LIN {X 0,Y 418.31,Z 399.821,A -85,B 0,C 180,E1 -10290.267,E2 -10290.267} C_VEL
LIN {X 0,Y 417.846,Z 405.193,A -85,B 0,C 180,E1 -10291.993,E2 -10291.993} C_VEL
LIN {X 0,Y 417.536,Z 409.039,A -85,B 0,C 180,E1 -10293.742,E2 -10293.742} C_VEL
LIN {X 0,Y 417.376,Z 410.854,A -85,B 0,C 180,E1 -10294.925,E2 -10294.925} C_VEL
LIN {X 0,Y 417.277,Z 412.013,A -85,B 0,C 180,E1 -10296.121,E2 -10296.121} C_VEL
LIN {X 0,Y 417.19,Z 412.615,A -85,B 0,C 180,E1 -10297.65,E2 -10297.65} C_VEL
LIN {X 0,Y 417.218,Z 412.19,A -85,B 0,C 180,E1 -10299.207,E2 -10299.207} C_VEL
LIN {X 0,Y 417.254,Z 410.33,A -85,B 0,C 180,E1 -10301.064,E2 -10301.064} C_VEL
LIN {X 0,Y 417.561,Z 406.754,A -85,B 0,C 180,E1 -10302.973,E2 -10302.973} C_VEL
LIN {X 0,Y 417.802,Z 402.306,A -85,B 0,C 180,E1 -10304.611,E2 -10304.611} C_VEL
LIN {X 0,Y 418.147,Z 396.207,A -85,B 0,C 180,E1 -10306.28,E2 -10306.28} C_VEL
LIN {X 0,Y 418.601,Z 389.043,A -85,B 0,C 180,E1 -10307.812,E2 -10307.812} C_VEL
LIN {X 0,Y 419.168,Z 381.176,A -85,B 0,C 180,E1 -10309.164,E2 -10309.164} C_VEL
LIN {X 0,Y 419.798,Z 371.573,A -85,B 0,C 180,E1 -10310.493,E2 -10310.493} C_VEL
LIN {X 0,Y 420.433,Z 361.16,A -85,B 0,C 180,E1 -10311.657,E2 -10311.657} C_VEL
LIN {X 0,Y 421.113,Z 349.41,A -85,B 0,C 180,E1 -10312.698,E2 -10312.698} C_VEL
LIN {X 0,Y 421.702,Z 337.687,A -85,B 0,C 180,E1 -10313.505,E2 -10313.505} C_VEL
LIN {X 0,Y 422.117,Z 325.639,A -85,B 0,C 180,E1 -10314.137,E2 -10314.137} C_VEL
LIN {X 0,Y 422.396,Z 313.572,A -85,B 0,C 180,E1 -10314.588,E2 -10314.588} C_VEL
LIN {X 0,Y 422.59,Z 300.07,A -85,B 0,C 180,E1 -10314.896,E2 -10314.896} C_VEL
LIN {X 0,Y 423.699,Z 218.43,A -85,B 0,C 180,E1 -10316.385,E2 -10316.385} C_VEL
LIN {X 0,Y 418.788,Z 204.246,A -85,B 0,C 180,E1 -10316.864,E2 -10316.864} C_VEL
LIN {X 0,Y 418.263,Z 202.387,A -85,B 0,C 180,E1 -10316.944,E2 -10316.944} C_VEL
LIN {X 0,Y 418.244,Z 202.385,A -85,B 0,C 180,E1 -10319.728,E2 -10319.728} C_VEL
LIN {X 0,Y 418.305,Z 202.381,A -85,B 0,C 180,E1 -10323.023,E2 -10323.023} C_VEL
LIN {X 0,Y 418.273,Z 202.379,A -85,B 0,C 180,E1 -10326.218,E2 -10326.218} C_VEL
LIN {X 0,Y 418.232,Z 202.385,A -85,B 0,C 180,E1 -10328.246,E2 -10328.246} C_VEL
LIN {X 0,Y 417.595,Z 202.47,A -85,B 0,C 180,E1 -10329.05,E2 -10329.05} C_VEL
LIN {X 0,Y 414.761,Z 202.818,A -85,B 0,C 180,E1 -10330.357,E2 -10330.357} C_VEL
LIN {X 0,Y 412.349,Z 203.119,A -85,B 0,C 180,E1 -10331.413,E2 -10331.413} C_VEL
LIN {X 0,Y 411.316,Z 203.246,A -85,B 0,C 180,E1 -10332.229,E2 -10332.229} C_VEL
LIN {X 0,Y 411.235,Z 203.256,A -85,B 0,C 180,E1 -10332.505,E2 -10332.505} C_VEL
LIN {X 0,Y 411.26,Z 203.256,A -85,B 0,C 180,E1 -10335.148,E2 -10335.148} C_VEL
LIN {X 0,Y 411.285,Z 203.251,A -85,B 0,C 180,E1 -10338.168,E2 -10338.168} C_VEL
LIN {X 0,Y 411.32,Z 203.248,A -85,B 0,C 180,E1 -10341.154,E2 -10341.154} C_VEL
LIN {X 0,Y 411.445,Z 203.231,A -85,B 0,C 180,E1 -10344.118,E2 -10344.118} C_VEL
LIN {X 0,Y 411.511,Z 203.223,A -85,B 0,C 180,E1 -10348.043,E2 -10348.043} C_VEL
LIN {X 0,Y 411.637,Z 203.208,A -85,B 0,C 180,E1 -10350,E2 -10350} C_VEL
LIN {X 0,Y 411.446,Z 203.231,A -85,B 0,C 180,E1 -10352.938,E2 -10352.938} C_VEL
LIN {X 0,Y 411.425,Z 203.234,A -85,B 0,C 180,E1 -10356.868,E2 -10356.868} C_VEL
LIN {X 0,Y 411.293,Z 203.251,A -85,B 0,C 180,E1 -10359.839,E2 -10359.839} C_VEL
LIN {X 0,Y 411.307,Z 203.247,A -85,B 0,C 180,E1 -10363.104,E2 -10363.104} C_VEL
LIN {X 0,Y 411.259,Z 203.253,A -85,B 0,C 180,E1 -10366.889,E2 -10366.889} C_VEL
LIN {X 0,Y 411.233,Z 203.263,A -85,B 0,C 180,E1 -10369.987,E2 -10369.987} C_VEL
LIN {X 0,Y 411.197,Z 203.261,A -85,B 0,C 180,E1 -10373.148,E2 -10373.148} C_VEL
LIN {X 0,Y 411.197,Z 203.262,A -85,B 0,C 180,E1 -10376.384,E2 -10376.384} C_VEL
LIN {X 0,Y 411.2,Z 203.266,A -85,B 0,C 180,E1 -10379.713,E2 -10379.713} C_VEL
LIN {X 0,Y 411.209,Z 203.261,A -85,B 0,C 180,E1 -10383.156,E2 -10383.156} C_VEL
LIN {X 0,Y 411.194,Z 203.261,A -85,B 0,C 180,E1 -10386.553,E2 -10386.553} C_VEL
LIN {X 0,Y 411.194,Z 203.266,A -85,B 0,C 180,E1 -10389.724,E2 -10389.724} C_VEL
LIN {X 0,Y 411.172,Z 203.267,A -85,B 0,C 180,E1 -10393.134,E2 -10393.134} C_VEL
LIN {X 0,Y 411.169,Z 203.266,A -85,B 0,C 180,E1 -10395.881,E2 -10395.881} C_VEL
LIN {X 0,Y 411.154,Z 203.267,A -85,B 0,C 180,E1 -10398.774,E2 -10398.774} C_VEL
LIN {X 0,Y 411.188,Z 203.262,A -85,B 0,C 180,E1 -10402.026,E2 -10402.026} C_VEL
LIN {X 0,Y 411.207,Z 203.261,A -85,B 0,C 180,E1 -10405.667,E2 -10405.667} C_VEL
LIN {X 0,Y 411.191,Z 203.268,A -85,B 0,C 180,E1 -10409.153,E2 -10409.153} C_VEL
LIN {X 0,Y 411.182,Z 203.265,A -85,B 0,C 180,E1 -10411.407,E2 -10411.407} C_VEL
LIN {X 0,Y 411.229,Z 203.264,A -85,B 0,C 180,E1 -10414.93,E2 -10414.93} C_VEL
LIN {X 0,Y 411.207,Z 203.259,A -85,B 0,C 180,E1 -10417.914,E2 -10417.914} C_VEL
LIN {X 0,Y 411.222,Z 203.262,A -85,B 0,C 180,E1 -10421.051,E2 -10421.051} C_VEL
LIN {X 0,Y 411.256,Z 203.254,A -85,B 0,C 180,E1 -10424.132,E2 -10424.132} C_VEL
LIN {X 0,Y 411.306,Z 203.249,A -85,B 0,C 180,E1 -10427.166,E2 -10427.166} C_VEL
LIN {X 0,Y 411.293,Z 203.251,A -85,B 0,C 180,E1 -10430.161,E2 -10430.161} C_VEL
LIN {X 0,Y 411.396,Z 203.237,A -85,B 0,C 180,E1 -10433.132,E2 -10433.132} C_VEL
LIN {X 0,Y 411.301,Z 203.249,A -85,B 0,C 180,E1 -10435.099,E2 -10435.099} C_VEL
LIN {X 0,Y 411.512,Z 203.224,A -85,B 0,C 180,E1 -10438.043,E2 -10438.043} C_VEL
LIN {X 0,Y 411.433,Z 203.232,A -85,B 0,C 180,E1 -10440.979,E2 -10440.979} C_VEL
LIN {X 0,Y 411.433,Z 203.232,A -85,B 0,C 180,E1 -10442.938,E2 -10442.938} C_VEL
LIN {X 0,Y 411.432,Z 203.234,A -85,B 0,C 180,E1 -10445.883,E2 -10445.883} C_VEL
LIN {X 0,Y 411.32,Z 203.246,A -85,B 0,C 180,E1 -10448.846,E2 -10448.846} C_VEL
LIN {X 0,Y 411.286,Z 203.254,A -85,B 0,C 180,E1 -10451.833,E2 -10451.833} C_VEL
LIN {X 0,Y 411.235,Z 203.256,A -85,B 0,C 180,E1 -10454.854,E2 -10454.854} C_VEL
LIN {X 0,Y 411.233,Z 203.263,A -85,B 0,C 180,E1 -10457.916,E2 -10457.916} C_VEL
LIN {X 0,Y 411.199,Z 203.26,A -85,B 0,C 180,E1 -10461.034,E2 -10461.034} C_VEL
LIN {X 0,Y 411.195,Z 203.263,A -85,B 0,C 180,E1 -10464.218,E2 -10464.218} C_VEL
LIN {X 0,Y 411.175,Z 203.268,A -85,B 0,C 180,E1 -10467.484,E2 -10467.484} C_VEL
LIN {X 0,Y 411.2,Z 203.267,A -85,B 0,C 180,E1 -10469.713,E2 -10469.713} C_VEL
LIN {X 0,Y 411.207,Z 203.262,A -85,B 0,C 180,E1 -10473.156,E2 -10473.156} C_VEL
LIN {X 0,Y 411.194,Z 203.261,A -85,B 0,C 180,E1 -10476.552,E2 -10476.552} C_VEL
LIN {X 0,Y 411.172,Z 203.267,A -85,B 0,C 180,E1 -10479.72,E2 -10479.72} C_VEL
LIN {X 0,Y 411.165,Z 203.269,A -85,B 0,C 180,E1 -10483.135,E2 -10483.135} C_VEL
LIN {X 0,Y 411.166,Z 203.266,A -85,B 0,C 180,E1 -10485.882,E2 -10485.882} C_VEL
LIN {X 0,Y 411.165,Z 203.268,A -85,B 0,C 180,E1 -10489.493,E2 -10489.493} C_VEL
LIN {X 0,Y 411.19,Z 203.262,A -85,B 0,C 180,E1 -10492.025,E2 -10492.025} C_VEL
LIN {X 0,Y 411.195,Z 203.263,A -85,B 0,C 180,E1 -10495.665,E2 -10495.665} C_VEL
LIN {X 0,Y 411.191,Z 203.267,A -85,B 0,C 180,E1 -10499.152,E2 -10499.152} C_VEL
LIN {X 0,Y 411.262,Z 203.344,A -85,B 0,C 180,E1 -10500.374,E2 -10500.374} C_VEL
LIN {X 0,Y 414.279,Z 218.043,A -85,B 0,C 180,E1 -10503.284,E2 -10503.284} C_VEL
LIN {X 0,Y 414.784,Z 222.006,A -85,B 0,C 180,E1 -10504.037,E2 -10504.037} C_VEL
LIN {X 0,Y 413.508,Z 241.529,A -85,B 0,C 180,E1 -10507.517,E2 -10507.517} C_VEL
LIN {X 0,Y 412.396,Z 260.082,A -85,B 0,C 180,E1 -10510.784,E2 -10510.784} C_VEL
LIN {X 0,Y 416.32,Z 291.809,A -85,B 0,C 180,E1 -10511.587,E2 -10511.587} C_VEL
LIN {X 0,Y 415.21,Z 369.766,A -85,B 0,C 180,E1 -10513.055,E2 -10513.055} C_VEL
LIN {X 0,Y 414.703,Z 383.404,A -85,B 0,C 180,E1 -10513.509,E2 -10513.509} C_VEL
LIN {X 0,Y 414.037,Z 395.804,A -85,B 0,C 180,E1 -10514.114,E2 -10514.114} C_VEL
LIN {X 0,Y 413.33,Z 406.944,A -85,B 0,C 180,E1 -10514.845,E2 -10514.845} C_VEL
LIN {X 0,Y 412.607,Z 417.276,A -85,B 0,C 180,E1 -10515.701,E2 -10515.701} C_VEL
LIN {X 0,Y 411.914,Z 428.377,A -85,B 0,C 180,E1 -10516.85,E2 -10516.85} C_VEL
LIN {X 0,Y 411.315,Z 438.558,A -85,B 0,C 180,E1 -10518.168,E2 -10518.168} C_VEL
LIN {X 0,Y 410.671,Z 447.696,A -85,B 0,C 180,E1 -10519.648,E2 -10519.648} C_VEL
LIN {X 0,Y 410.341,Z 455.065,A -85,B 0,C 180,E1 -10521.133,E2 -10521.133} C_VEL
LIN {X 0,Y 410.171,Z 460.941,A -85,B 0,C 180,E1 -10522.616,E2 -10522.616} C_VEL
LIN {X 0,Y 410.066,Z 465.54,A -85,B 0,C 180,E1 -10524.097,E2 -10524.097} C_VEL
LIN {X 0,Y 410.102,Z 467.957,A -85,B 0,C 180,E1 -10525.084,E2 -10525.084} C_VEL
LIN {X 0,Y 410.061,Z 469.921,A -85,B 0,C 180,E1 -10526.069,E2 -10526.069} C_VEL
LIN {X 0,Y 410.17,Z 471.461,A -85,B 0,C 180,E1 -10527.053,E2 -10527.053} C_VEL
LIN {X 0,Y 410.173,Z 472.52,A -85,B 0,C 180,E1 -10528.036,E2 -10528.036} C_VEL
LIN {X 0,Y 410.163,Z 473.165,A -85,B 0,C 180,E1 -10529.018,E2 -10529.018} C_VEL
LIN {X 0,Y 410.14,Z 473.407,A -85,B 0,C 180,E1 -10530,E2 -10530} C_VEL
LIN {X 0,Y 410.163,Z 473.239,A -85,B 0,C 180,E1 -10530.982,E2 -10530.982} C_VEL
LIN {X 0,Y 410.15,Z 472.618,A -85,B 0,C 180,E1 -10531.964,E2 -10531.964} C_VEL
LIN {X 0,Y 410.174,Z 471.595,A -85,B 0,C 180,E1 -10532.946,E2 -10532.946} C_VEL
LIN {X 0,Y 410.06,Z 470.15,A -85,B 0,C 180,E1 -10533.931,E2 -10533.931} C_VEL
LIN {X 0,Y 410.08,Z 467.14,A -85,B 0,C 180,E1 -10535.408,E2 -10535.408} C_VEL
LIN {X 0,Y 410.162,Z 463.07,A -85,B 0,C 180,E1 -10536.889,E2 -10536.889} C_VEL
LIN {X 0,Y 410.336,Z 456.838,A -85,B 0,C 180,E1 -10538.619,E2 -10538.619} C_VEL
LIN {X 0,Y 410.617,Z 450.013,A -85,B 0,C 180,E1 -10540.104,E2 -10540.104} C_VEL
LIN {X 0,Y 411.22,Z 441.574,A -85,B 0,C 180,E1 -10541.584,E2 -10541.584} C_VEL
LIN {X 0,Y 411.787,Z 432.967,A -85,B 0,C 180,E1 -10542.819,E2 -10542.819} C_VEL
LIN {X 0,Y 412.572,Z 422.411,A -85,B 0,C 180,E1 -10544.048,E2 -10544.048} C_VEL
LIN {X 0,Y 413.448,Z 410.573,A -85,B 0,C 180,E1 -10545.15,E2 -10545.15} C_VEL
LIN {X 0,Y 414.331,Z 398.849,A -85,B 0,C 180,E1 -10546,E2 -10546} C_VEL
LIN {X 0,Y 415.062,Z 386.782,A -85,B 0,C 180,E1 -10546.666,E2 -10546.666} C_VEL
LIN {X 0,Y 415.84,Z 372.978,A -85,B 0,C 180,E1 -10547.203,E2 -10547.203} C_VEL
LIN {X 0,Y 416.177,Z 358.822,A -85,B 0,C 180,E1 -10547.537,E2 -10547.537} C_VEL
LIN {X 0,Y 417.102,Z 289.747,A -85,B 0,C 180,E1 -10548.852,E2 -10548.852} C_VEL
LIN {X 0,Y 414.27,Z 267.739,A -85,B 0,C 180,E1 -10549.447,E2 -10549.447} C_VEL
LIN {X 0,Y 412.657,Z 257.23,A -85,B 0,C 180,E1 -10549.78,E2 -10549.78} C_VEL
LIN {X 0,Y 413.871,Z 235.468,A -85,B 0,C 180,E1 -10553.511,E2 -10553.511} C_VEL
LIN {X 0,Y 414.745,Z 220.411,A -85,B 0,C 180,E1 -10556.141,E2 -10556.141} C_VEL
LIN {X 0,Y 412.639,Z 209.36,A -85,B 0,C 180,E1 -10558.274,E2 -10558.274} C_VEL
LIN {X 0,Y 411.211,Z 203.268,A -85,B 0,C 180,E1 -10559.54,E2 -10559.54} C_VEL
LIN {X 0,Y 411.207,Z 203.265,A -85,B 0,C 180,E1 -10563.155,E2 -10563.155} C_VEL
LIN {X 0,Y 411.192,Z 203.267,A -85,B 0,C 180,E1 -10566.552,E2 -10566.552} C_VEL
LIN {X 0,Y 411.17,Z 203.266,A -85,B 0,C 180,E1 -10569.72,E2 -10569.72} C_VEL
LIN {X 0,Y 411.17,Z 203.266,A -85,B 0,C 180,E1 -10573.134,E2 -10573.134} C_VEL
LIN {X 0,Y 411.167,Z 203.265,A -85,B 0,C 180,E1 -10575.881,E2 -10575.881} C_VEL
LIN {X 0,Y 411.155,Z 203.27,A -85,B 0,C 180,E1 -10578.773,E2 -10578.773} C_VEL
LIN {X 0,Y 411.186,Z 203.266,A -85,B 0,C 180,E1 -10582.025,E2 -10582.025} C_VEL
LIN {X 0,Y 411.205,Z 203.26,A -85,B 0,C 180,E1 -10585.666,E2 -10585.666} C_VEL
LIN {X 0,Y 411.189,Z 203.263,A -85,B 0,C 180,E1 -10589.152,E2 -10589.152} C_VEL
LIN {X 0,Y 411.189,Z 203.263,A -85,B 0,C 180,E1 -10592.517,E2 -10592.517} C_VEL
LIN {X 0,Y 411.211,Z 203.264,A -85,B 0,C 180,E1 -10595.784,E2 -10595.784} C_VEL
LIN {X 0,Y 411.196,Z 203.261,A -85,B 0,C 180,E1 -10598.966,E2 -10598.966} C_VEL
LIN {X 0,Y 411.245,Z 203.256,A -85,B 0,C 180,E1 -10602.084,E2 -10602.084} C_VEL
LIN {X 0,Y 411.258,Z 203.254,A -85,B 0,C 180,E1 -10605.147,E2 -10605.147} C_VEL
LIN {X 0,Y 411.283,Z 203.25,A -85,B 0,C 180,E1 -10608.167,E2 -10608.167} C_VEL
LIN {X 0,Y 411.44,Z 203.233,A -85,B 0,C 180,E1 -10612.189,E2 -10612.189} C_VEL
LIN {X 0,Y 411.471,Z 203.229,A -85,B 0,C 180,E1 -10614.118,E2 -10614.118} C_VEL
LIN {X 0,Y 411.51,Z 203.223,A -85,B 0,C 180,E1 -10618.042,E2 -10618.042} C_VEL
LIN {X 0,Y 411.64,Z 203.208,A -85,B 0,C 180,E1 -10620,E2 -10620} C_VEL
LIN {X 0,Y 411.458,Z 203.233,A -85,B 0,C 180,E1 -10622.937,E2 -10622.937} C_VEL
LIN {X 0,Y 411.424,Z 203.237,A -85,B 0,C 180,E1 -10626.868,E2 -10626.868} C_VEL
LIN {X 0,Y 411.291,Z 203.254,A -85,B 0,C 180,E1 -10629.839,E2 -10629.839} C_VEL
LIN {X 0,Y 411.305,Z 203.258,A -85,B 0,C 180,E1 -10633.104,E2 -10633.104} C_VEL
LIN {X 0,Y 411.302,Z 203.255,A -85,B 0,C 180,E1 -10636.887,E2 -10636.887} C_VEL
LIN {X 0,Y 411.275,Z 203.368,A -85,B 0,C 180,E1 -10638.089,E2 -10638.089} C_VEL
LIN {X 0,Y 411.383,Z 204.007,A -85,B 0,C 180,E1 -10638.23,E2 -10638.23} C_VEL
LIN {X 0,Y 418.004,Z 220.696,A -85,B 0,C 180,E1 -10638.962,E2 -10638.962} C_VEL
LIN {X 0,Y 418.199,Z 223.122,A -85,B 0,C 180,E1 -10639.023,E2 -10639.023} C_VEL
LIN {X 0,Y 416.618,Z 312.115,A -85,B 0,C 180,E1 -10640.748,E2 -10640.748} C_VEL
LIN {X 0,Y 416.297,Z 325.297,A -85,B 0,C 180,E1 -10641.207,E2 -10641.207} C_VEL
LIN {X 0,Y 415.811,Z 337.595,A -85,B 0,C 180,E1 -10641.829,E2 -10641.829} C_VEL
LIN {X 0,Y 415.142,Z 349.63,A -85,B 0,C 180,E1 -10642.652,E2 -10642.652} C_VEL
LIN {X 0,Y 414.418,Z 361.332,A -85,B 0,C 180,E1 -10643.685,E2 -10643.685} C_VEL
LIN {X 0,Y 413.704,Z 370.819,A -85,B 0,C 180,E1 -10644.729,E2 -10644.729} C_VEL
LIN {X 0,Y 412.924,Z 380.721,A -85,B 0,C 180,E1 -10646.087,E2 -10646.087} C_VEL
LIN {X 0,Y 412.225,Z 389.352,A -85,B 0,C 180,E1 -10647.558,E2 -10647.558} C_VEL
LIN {X 0,Y 411.657,Z 396.03,A -85,B 0,C 180,E1 -10648.981,E2 -10648.981} C_VEL
LIN {X 0,Y 411.257,Z 400.954,A -85,B 0,C 180,E1 -10650.273,E2 -10650.273} C_VEL
LIN {X 0,Y 410.787,Z 406.143,A -85,B 0,C 180,E1 -10652.03,E2 -10652.03} C_VEL
LIN {X 0,Y 410.565,Z 408.808,A -85,B 0,C 180,E1 -10653.214,E2 -10653.214} C_VEL
LIN {X 0,Y 410.338,Z 411.212,A -85,B 0,C 180,E1 -10654.703,E2 -10654.703} C_VEL
LIN {X 0,Y 410.175,Z 412.762,A -85,B 0,C 180,E1 -10656.361,E2 -10656.361} C_VEL
LIN {X 0,Y 410.105,Z 413.13,A -85,B 0,C 180,E1 -10658.093,E2 -10658.093} C_VEL
LIN {X 0,Y 410.128,Z 412.496,A -85,B 0,C 180,E1 -10659.545,E2 -10659.545} C_VEL
LIN {X 0,Y 410.191,Z 410.866,A -85,B 0,C 180,E1 -10661.073,E2 -10661.073} C_VEL
LIN {X 0,Y 410.412,Z 408.258,A -85,B 0,C 180,E1 -10662.579,E2 -10662.579} C_VEL
LIN {X 0,Y 410.649,Z 404.716,A -85,B 0,C 180,E1 -10664.045,E2 -10664.045} C_VEL
LIN {X 0,Y 410.942,Z 400.192,A -85,B 0,C 180,E1 -10665.478,E2 -10665.478} C_VEL
LIN {X 0,Y 411.284,Z 394.627,A -85,B 0,C 180,E1 -10666.881,E2 -10666.881} C_VEL
LIN {X 0,Y 411.798,Z 386.98,A -85,B 0,C 180,E1 -10668.42,E2 -10668.42} C_VEL
LIN {X 0,Y 412.467,Z 377.916,A -85,B 0,C 180,E1 -10669.882,E2 -10669.882} C_VEL
LIN {X 0,Y 413.124,Z 368.305,A -85,B 0,C 180,E1 -10671.124,E2 -10671.124} C_VEL
LIN {X 0,Y 413.776,Z 356.952,A -85,B 0,C 180,E1 -10672.305,E2 -10672.305} C_VEL
LIN {X 0,Y 414.44,Z 345.272,A -85,B 0,C 180,E1 -10673.259,E2 -10673.259} C_VEL
LIN {X 0,Y 415.006,Z 332.802,A -85,B 0,C 180,E1 -10674.038,E2 -10674.038} C_VEL
LIN {X 0,Y 415.376,Z 319.704,A -85,B 0,C 180,E1 -10674.639,E2 -10674.639} C_VEL
LIN {X 0,Y 415.641,Z 306.409,A -85,B 0,C 180,E1 -10675.028,E2 -10675.028} C_VEL
LIN {X 0,Y 416.95,Z 219.897,A -85,B 0,C 180,E1 -10676.639,E2 -10676.639} C_VEL
LIN {X 0,Y 411.947,Z 205.622,A -85,B 0,C 180,E1 -10677.135,E2 -10677.135} C_VEL
LIN {X 0,Y 411.235,Z 203.263,A -85,B 0,C 180,E1 -10677.23,E2 -10677.23} C_VEL
LIN {X 0,Y 411.233,Z 203.259,A -85,B 0,C 180,E1 -10680.644,E2 -10680.644} C_VEL
LIN {X 0,Y 411.233,Z 203.258,A -85,B 0,C 180,E1 -10683.619,E2 -10683.619} C_VEL
LIN {X 0,Y 411.195,Z 203.265,A -85,B 0,C 180,E1 -10686.852,E2 -10686.852} C_VEL
LIN {X 0,Y 411.215,Z 203.258,A -85,B 0,C 180,E1 -10690.051,E2 -10690.051} C_VEL
LIN {X 0,Y 411.235,Z 203.256,A -85,B 0,C 180,E1 -10692.505,E2 -10692.505} C_VEL
LIN {X 0,Y 410.568,Z 203.344,A -85,B 0,C 180,E1 -10693.322,E2 -10693.322} C_VEL
LIN {X 0,Y 407.703,Z 203.707,A -85,B 0,C 180,E1 -10694.65,E2 -10694.65} C_VEL
LIN {X 0,Y 405.309,Z 204.006,A -85,B 0,C 180,E1 -10695.723,E2 -10695.723} C_VEL
LIN {X 0,Y 404.327,Z 204.125,A -85,B 0,C 180,E1 -10696.553,E2 -10696.553} C_VEL
LIN {X 0,Y 404.272,Z 204.13,A -85,B 0,C 180,E1 -10696.833,E2 -10696.833} C_VEL
LIN {X 0,Y 404.258,Z 204.125,A -85,B 0,C 180,E1 -10699.989,E2 -10699.989} C_VEL
LIN {X 0,Y 404.371,Z 204.114,A -85,B 0,C 180,E1 -10703.012,E2 -10703.012} C_VEL
LIN {X 0,Y 404.276,Z 204.125,A -85,B 0,C 180,E1 -10705.014,E2 -10705.014} C_VEL
LIN {X 0,Y 404.48,Z 204.099,A -85,B 0,C 180,E1 -10708.009,E2 -10708.009} C_VEL
LIN {X 0,Y 404.607,Z 204.083,A -85,B 0,C 180,E1 -10710,E2 -10710} C_VEL
LIN {X 0,Y 404.404,Z 204.108,A -85,B 0,C 180,E1 -10712.989,E2 -10712.989} C_VEL
LIN {X 0,Y 404.371,Z 204.112,A -85,B 0,C 180,E1 -10716.988,E2 -10716.988} C_VEL
LIN {X 0,Y 404.258,Z 204.129,A -85,B 0,C 180,E1 -10720.012,E2 -10720.012} C_VEL
LIN {X 0,Y 404.268,Z 204.124,A -85,B 0,C 180,E1 -10723.212,E2 -10723.212} C_VEL
LIN {X 0,Y 404.218,Z 204.13,A -85,B 0,C 180,E1 -10727.007,E2 -10727.007} C_VEL
LIN {X 0,Y 404.166,Z 204.14,A -85,B 0,C 180,E1 -10730.352,E2 -10730.352} C_VEL
LIN {X 0,Y 404.162,Z 204.14,A -85,B 0,C 180,E1 -10733.575,E2 -10733.575} C_VEL
LIN {X 0,Y 404.136,Z 204.14,A -85,B 0,C 180,E1 -10736.882,E2 -10736.882} C_VEL
LIN {X 0,Y 404.146,Z 204.141,A -85,B 0,C 180,E1 -10740.285,E2 -10740.285} C_VEL
LIN {X 0,Y 404.147,Z 204.145,A -85,B 0,C 180,E1 -10743.812,E2 -10743.812} C_VEL
LIN {X 0,Y 404.136,Z 204.141,A -85,B 0,C 180,E1 -10746.875,E2 -10746.875} C_VEL
LIN {X 0,Y 404.15,Z 204.14,A -85,B 0,C 180,E1 -10750.08,E2 -10750.08} C_VEL
LIN {X 0,Y 404.152,Z 204.141,A -85,B 0,C 180,E1 -10753.083,E2 -10753.083} C_VEL
LIN {X 0,Y 404.149,Z 204.14,A -85,B 0,C 180,E1 -10755.926,E2 -10755.926} C_VEL
LIN {X 0,Y 404.11,Z 204.144,A -85,B 0,C 180,E1 -10758.634,E2 -10758.634} C_VEL
LIN {X 0,Y 404.142,Z 204.144,A -85,B 0,C 180,E1 -10761.495,E2 -10761.495} C_VEL
LIN {X 0,Y 404.186,Z 204.138,A -85,B 0,C 180,E1 -10764.984,E2 -10764.984} C_VEL
LIN {X 0,Y 404.144,Z 204.141,A -85,B 0,C 180,E1 -10768.554,E2 -10768.554} C_VEL
LIN {X 0,Y 404.155,Z 204.143,A -85,B 0,C 180,E1 -10770.863,E2 -10770.863} C_VEL
LIN {X 0,Y 404.149,Z 204.139,A -85,B 0,C 180,E1 -10774.231,E2 -10774.231} C_VEL
LIN {X 0,Y 404.171,Z 204.137,A -85,B 0,C 180,E1 -10777.508,E2 -10777.508} C_VEL
LIN {X 0,Y 404.165,Z 204.142,A -85,B 0,C 180,E1 -10780.708,E2 -10780.708} C_VEL
LIN {X 0,Y 404.223,Z 204.129,A -85,B 0,C 180,E1 -10783.848,E2 -10783.848} C_VEL
LIN {X 0,Y 404.286,Z 204.125,A -85,B 0,C 180,E1 -10786.939,E2 -10786.939} C_VEL
LIN {X 0,Y 404.259,Z 204.126,A -85,B 0,C 180,E1 -10789.988,E2 -10789.988} C_VEL
LIN {X 0,Y 404.346,Z 204.116,A -85,B 0,C 180,E1 -10793.012,E2 -10793.012} C_VEL
LIN {X 0,Y 404.272,Z 204.125,A -85,B 0,C 180,E1 -10795.014,E2 -10795.014} C_VEL
LIN {X 0,Y 404.48,Z 204.1,A -85,B 0,C 180,E1 -10798.009,E2 -10798.009} C_VEL
LIN {X 0,Y 404.398,Z 204.108,A -85,B 0,C 180,E1 -10800.996,E2 -10800.996} C_VEL
LIN {X 0,Y 404.392,Z 204.109,A -85,B 0,C 180,E1 -10802.989,E2 -10802.989} C_VEL
LIN {X 0,Y 404.38,Z 204.114,A -85,B 0,C 180,E1 -10805.986,E2 -10805.986} C_VEL
LIN {X 0,Y 404.267,Z 204.124,A -85,B 0,C 180,E1 -10809.002,E2 -10809.002} C_VEL
LIN {X 0,Y 404.259,Z 204.132,A -85,B 0,C 180,E1 -10812.042,E2 -10812.042} C_VEL
LIN {X 0,Y 404.179,Z 204.135,A -85,B 0,C 180,E1 -10815.119,E2 -10815.119} C_VEL
LIN {X 0,Y 404.197,Z 204.136,A -85,B 0,C 180,E1 -10818.239,E2 -10818.239} C_VEL
LIN {X 0,Y 404.141,Z 204.142,A -85,B 0,C 180,E1 -10821.419,E2 -10821.419} C_VEL
LIN {X 0,Y 404.151,Z 204.138,A -85,B 0,C 180,E1 -10824.667,E2 -10824.667} C_VEL
LIN {X 0,Y 404.118,Z 204.146,A -85,B 0,C 180,E1 -10828.006,E2 -10828.006} C_VEL
LIN {X 0,Y 404.146,Z 204.14,A -85,B 0,C 180,E1 -10830.285,E2 -10830.285} C_VEL
LIN {X 0,Y 404.141,Z 204.144,A -85,B 0,C 180,E1 -10833.813,E2 -10833.813} C_VEL
LIN {X 0,Y 404.137,Z 204.141,A -85,B 0,C 180,E1 -10836.874,E2 -10836.874} C_VEL
LIN {X 0,Y 404.119,Z 204.143,A -85,B 0,C 180,E1 -10840.075,E2 -10840.075} C_VEL
LIN {X 0,Y 404.144,Z 204.143,A -85,B 0,C 180,E1 -10843.082,E2 -10843.082} C_VEL
LIN {X 0,Y 404.123,Z 204.143,A -85,B 0,C 180,E1 -10845.922,E2 -10845.922} C_VEL
LIN {X 0,Y 404.105,Z 204.145,A -85,B 0,C 180,E1 -10848.633,E2 -10848.633} C_VEL
LIN {X 0,Y 404.144,Z 204.142,A -85,B 0,C 180,E1 -10851.494,E2 -10851.494} C_VEL
LIN {X 0,Y 404.176,Z 204.141,A -85,B 0,C 180,E1 -10854.983,E2 -10854.983} C_VEL
LIN {X 0,Y 404.139,Z 204.144,A -85,B 0,C 180,E1 -10858.442,E2 -10858.442} C_VEL
LIN {X 0,Y 404.209,Z 204.231,A -85,B 0,C 180,E1 -10860.122,E2 -10860.122} C_VEL
LIN {X 0,Y 407.21,Z 218.794,A -85,B 0,C 180,E1 -10863.06,E2 -10863.06} C_VEL
LIN {X 0,Y 407.807,Z 223.769,A -85,B 0,C 180,E1 -10864.02,E2 -10864.02} C_VEL
LIN {X 0,Y 406.523,Z 242.3,A -85,B 0,C 180,E1 -10867.377,E2 -10867.377} C_VEL
LIN {X 0,Y 405.471,Z 259.896,A -85,B 0,C 180,E1 -10870.509,E2 -10870.509} C_VEL
LIN {X 0,Y 409.506,Z 292.119,A -85,B 0,C 180,E1 -10871.322,E2 -10871.322} C_VEL
LIN {X 0,Y 408.387,Z 368.941,A -85,B 0,C 180,E1 -10872.795,E2 -10872.795} C_VEL
LIN {X 0,Y 407.84,Z 382.665,A -85,B 0,C 180,E1 -10873.255,E2 -10873.255} C_VEL
LIN {X 0,Y 407.097,Z 395.655,A -85,B 0,C 180,E1 -10873.901,E2 -10873.901} C_VEL
LIN {X 0,Y 406.309,Z 407.5,A -85,B 0,C 180,E1 -10874.705,E2 -10874.705} C_VEL
LIN {X 0,Y 405.489,Z 418.947,A -85,B 0,C 180,E1 -10875.701,E2 -10875.701} C_VEL
LIN {X 0,Y 404.877,Z 428.536,A -85,B 0,C 180,E1 -10876.738,E2 -10876.738} C_VEL
LIN {X 0,Y 404.269,Z 437.775,A -85,B 0,C 180,E1 -10877.959,E2 -10877.959} C_VEL
LIN {X 0,Y 403.65,Z 446.967,A -85,B 0,C 180,E1 -10879.466,E2 -10879.466} C_VEL
LIN {X 0,Y 403.29,Z 454.376,A -85,B 0,C 180,E1 -10880.976,E2 -10880.976} C_VEL
LIN {X 0,Y 403.097,Z 460.295,A -85,B 0,C 180,E1 -10882.486,E2 -10882.486} C_VEL
LIN {X 0,Y 402.99,Z 464.928,A -85,B 0,C 180,E1 -10883.993,E2 -10883.993} C_VEL
LIN {X 0,Y 403.033,Z 467.362,A -85,B 0,C 180,E1 -10884.998,E2 -10884.998} C_VEL
LIN {X 0,Y 402.974,Z 469.337,A -85,B 0,C 180,E1 -10885.999,E2 -10885.999} C_VEL
LIN {X 0,Y 403.1,Z 470.895,A -85,B 0,C 180,E1 -10887.002,E2 -10887.002} C_VEL
LIN {X 0,Y 403.095,Z 471.97,A -85,B 0,C 180,E1 -10888.001,E2 -10888.001} C_VEL
LIN {X 0,Y 403.109,Z 472.628,A -85,B 0,C 180,E1 -10889.001,E2 -10889.001} C_VEL
LIN {X 0,Y 403.084,Z 472.877,A -85,B 0,C 180,E1 -10890,E2 -10890} C_VEL
LIN {X 0,Y 403.091,Z 472.721,A -85,B 0,C 180,E1 -10890.999,E2 -10890.999} C_VEL
LIN {X 0,Y 403.075,Z 472.112,A -85,B 0,C 180,E1 -10891.998,E2 -10891.998} C_VEL
LIN {X 0,Y 403.085,Z 471.093,A -85,B 0,C 180,E1 -10892.998,E2 -10892.998} C_VEL
LIN {X 0,Y 402.972,Z 469.654,A -85,B 0,C 180,E1 -10894,E2 -10894} C_VEL
LIN {X 0,Y 402.975,Z 466.655,A -85,B 0,C 180,E1 -10895.504,E2 -10895.504} C_VEL
LIN {X 0,Y 403.072,Z 462.596,A -85,B 0,C 180,E1 -10897.01,E2 -10897.01} C_VEL
LIN {X 0,Y 403.265,Z 456.385,A -85,B 0,C 180,E1 -10898.771,E2 -10898.771} C_VEL
LIN {X 0,Y 403.563,Z 449.589,A -85,B 0,C 180,E1 -10900.282,E2 -10900.282} C_VEL
LIN {X 0,Y 404.232,Z 441.193,A -85,B 0,C 180,E1 -10901.787,E2 -10901.787} C_VEL
LIN {X 0,Y 404.942,Z 431.481,A -85,B 0,C 180,E1 -10903.193,E2 -10903.193} C_VEL
LIN {X 0,Y 405.741,Z 420.948,A -85,B 0,C 180,E1 -10904.418,E2 -10904.418} C_VEL
LIN {X 0,Y 406.593,Z 410.357,A -85,B 0,C 180,E1 -10905.412,E2 -10905.412} C_VEL
LIN {X 0,Y 407.515,Z 398.76,A -85,B 0,C 180,E1 -10906.275,E2 -10906.275} C_VEL
LIN {X 0,Y 408.277,Z 386.842,A -85,B 0,C 180,E1 -10906.951,E2 -10906.951} C_VEL
LIN {X 0,Y 409.071,Z 373.299,A -85,B 0,C 180,E1 -10907.497,E2 -10907.497} C_VEL
LIN {X 0,Y 409.479,Z 359.927,A -85,B 0,C 180,E1 -10907.834,E2 -10907.834} C_VEL
LIN {X 0,Y 410.46,Z 290.551,A -85,B 0,C 180,E1 -10909.183,E2 -10909.183} C_VEL
LIN {X 0,Y 407.784,Z 269.314,A -85,B 0,C 180,E1 -10909.775,E2 -10909.775} C_VEL
LIN {X 0,Y 405.806,Z 256.57,A -85,B 0,C 180,E1 -10910.188,E2 -10910.188} C_VEL
LIN {X 0,Y 407.021,Z 236.07,A -85,B 0,C 180,E1 -10913.773,E2 -10913.773} C_VEL
LIN {X 0,Y 407.858,Z 221.55,A -85,B 0,C 180,E1 -10916.358,E2 -10916.358} C_VEL
LIN {X 0,Y 405.417,Z 209.423,A -85,B 0,C 180,E1 -10918.759,E2 -10918.759} C_VEL
LIN {X 0,Y 404.156,Z 204.147,A -85,B 0,C 180,E1 -10919.898,E2 -10919.898} C_VEL
LIN {X 0,Y 404.171,Z 204.141,A -85,B 0,C 180,E1 -10923.42,E2 -10923.42} C_VEL
LIN {X 0,Y 404.141,Z 204.142,A -85,B 0,C 180,E1 -10926.246,E2 -10926.246} C_VEL
LIN {X 0,Y 404.135,Z 204.144,A -85,B 0,C 180,E1 -10928.759,E2 -10928.759} C_VEL
LIN {X 0,Y 404.113,Z 204.144,A -85,B 0,C 180,E1 -10931.598,E2 -10931.598} C_VEL
LIN {X 0,Y 404.145,Z 204.143,A -85,B 0,C 180,E1 -10934.522,E2 -10934.522} C_VEL
LIN {X 0,Y 404.131,Z 204.14,A -85,B 0,C 180,E1 -10937.295,E2 -10937.295} C_VEL
LIN {X 0,Y 404.132,Z 204.141,A -85,B 0,C 180,E1 -10939.951,E2 -10939.951} C_VEL
LIN {X 0,Y 404.134,Z 204.143,A -85,B 0,C 180,E1 -10943.125,E2 -10943.125} C_VEL
LIN {X 0,Y 404.145,Z 204.144,A -85,B 0,C 180,E1 -10946.188,E2 -10946.188} C_VEL
LIN {X 0,Y 404.144,Z 204.143,A -85,B 0,C 180,E1 -10949.715,E2 -10949.715} C_VEL
LIN {X 0,Y 404.135,Z 204.139,A -85,B 0,C 180,E1 -10953.118,E2 -10953.118} C_VEL
LIN {X 0,Y 404.16,Z 204.138,A -85,B 0,C 180,E1 -10956.425,E2 -10956.425} C_VEL
LIN {X 0,Y 404.191,Z 204.135,A -85,B 0,C 180,E1 -10959.874,E2 -10959.874} C_VEL
LIN {X 0,Y 404.216,Z 204.129,A -85,B 0,C 180,E1 -10962.993,E2 -10962.993} C_VEL
LIN {X 0,Y 404.283,Z 204.123,A -85,B 0,C 180,E1 -10966.939,E2 -10966.939} C_VEL
LIN {X 0,Y 404.257,Z 204.128,A -85,B 0,C 180,E1 -10969.988,E2 -10969.988} C_VEL
LIN {X 0,Y 404.399,Z 204.111,A -85,B 0,C 180,E1 -10973.012,E2 -10973.012} C_VEL
LIN {X 0,Y 404.28,Z 204.126,A -85,B 0,C 180,E1 -10975.013,E2 -10975.013} C_VEL
LIN {X 0,Y 404.479,Z 204.099,A -85,B 0,C 180,E1 -10978.008,E2 -10978.008} C_VEL
LIN {X 0,Y 404.61,Z 204.084,A -85,B 0,C 180,E1 -10980,E2 -10980} C_VEL
LIN {X 0,Y 404.416,Z 204.11,A -85,B 0,C 180,E1 -10982.988,E2 -10982.988} C_VEL
LIN {X 0,Y 404.37,Z 204.117,A -85,B 0,C 180,E1 -10986.988,E2 -10986.988} C_VEL
LIN {X 0,Y 404.257,Z 204.13,A -85,B 0,C 180,E1 -10990.012,E2 -10990.012} C_VEL
LIN {X 0,Y 404.266,Z 204.135,A -85,B 0,C 180,E1 -10993.211,E2 -10993.211} C_VEL
LIN {X 0,Y 404.248,Z 204.132,A -85,B 0,C 180,E1 -10997.191,E2 -10997.191} C_VEL
LIN {X 0,Y 404.23,Z 204.201,A -85,B 0,C 180,E1 -10997.713,E2 -10997.713} C_VEL
LIN {X 0,Y 404.453,Z 205.174,A -85,B 0,C 180,E1 -10997.829,E2 -10997.829} C_VEL
LIN {X 0,Y 410.621,Z 220.143,A -85,B 0,C 180,E1 -10998.524,E2 -10998.524} C_VEL
LIN {X 0,Y 411.611,Z 222.864,A -85,B 0,C 180,E1 -10998.639,E2 -10998.639} C_VEL
LIN {X 0,Y 409.949,Z 312.251,A -85,B 0,C 180,E1 -11000.412,E2 -11000.412} C_VEL
LIN {X 0,Y 409.616,Z 324.987,A -85,B 0,C 180,E1 -11000.856,E2 -11000.856} C_VEL
LIN {X 0,Y 409.105,Z 338.128,A -85,B 0,C 180,E1 -11001.525,E2 -11001.525} C_VEL
LIN {X 0,Y 408.369,Z 350.435,A -85,B 0,C 180,E1 -11002.381,E2 -11002.381} C_VEL
LIN {X 0,Y 407.652,Z 361.388,A -85,B 0,C 180,E1 -11003.361,E2 -11003.361} C_VEL
LIN {X 0,Y 406.872,Z 371.531,A -85,B 0,C 180,E1 -11004.491,E2 -11004.491} C_VEL
LIN {X 0,Y 406.062,Z 381.221,A -85,B 0,C 180,E1 -11005.842,E2 -11005.842} C_VEL
LIN {X 0,Y 405.343,Z 389.517,A -85,B 0,C 180,E1 -11007.273,E2 -11007.273} C_VEL
LIN {X 0,Y 404.703,Z 396.653,A -85,B 0,C 180,E1 -11008.81,E2 -11008.81} C_VEL
LIN {X 0,Y 404.2,Z 402.075,A -85,B 0,C 180,E1 -11010.281,E2 -11010.281} C_VEL
LIN {X 0,Y 403.715,Z 407.115,A -85,B 0,C 180,E1 -11012.069,E2 -11012.069} C_VEL
LIN {X 0,Y 403.396,Z 410.716,A -85,B 0,C 180,E1 -11013.884,E2 -11013.884} C_VEL
LIN {X 0,Y 403.224,Z 412.303,A -85,B 0,C 180,E1 -11015.112,E2 -11015.112} C_VEL
LIN {X 0,Y 403.085,Z 413.455,A -85,B 0,C 180,E1 -11016.676,E2 -11016.676} C_VEL
LIN {X 0,Y 403.022,Z 413.605,A -85,B 0,C 180,E1 -11018.305,E2 -11018.305} C_VEL
LIN {X 0,Y 403.063,Z 412.474,A -85,B 0,C 180,E1 -11020.177,E2 -11020.177} C_VEL
LIN {X 0,Y 403.257,Z 409.686,A -85,B 0,C 180,E1 -11022.143,E2 -11022.143} C_VEL
LIN {X 0,Y 403.519,Z 406.759,A -85,B 0,C 180,E1 -11023.517,E2 -11023.517} C_VEL
LIN {X 0,Y 403.783,Z 402.792,A -85,B 0,C 180,E1 -11024.939,E2 -11024.939} C_VEL
LIN {X 0,Y 404.135,Z 396.636,A -85,B 0,C 180,E1 -11026.638,E2 -11026.638} C_VEL
LIN {X 0,Y 404.633,Z 389.803,A -85,B 0,C 180,E1 -11028.126,E2 -11028.126} C_VEL
LIN {X 0,Y 405.257,Z 381.783,A -85,B 0,C 180,E1 -11029.537,E2 -11029.537} C_VEL
LIN {X 0,Y 405.863,Z 372.839,A -85,B 0,C 180,E1 -11030.813,E2 -11030.813} C_VEL
LIN {X 0,Y 406.597,Z 361.791,A -85,B 0,C 180,E1 -11032.087,E2 -11032.087} C_VEL
LIN {X 0,Y 407.267,Z 351.007,A -85,B 0,C 180,E1 -11033.076,E2 -11033.076} C_VEL
LIN {X 0,Y 407.899,Z 339.473,A -85,B 0,C 180,E1 -11033.908,E2 -11033.908} C_VEL
LIN {X 0,Y 408.373,Z 327.53,A -85,B 0,C 180,E1 -11034.567,E2 -11034.567} C_VEL
LIN {X 0,Y 408.704,Z 315.333,A -85,B 0,C 180,E1 -11035.052,E2 -11035.052} C_VEL
LIN {X 0,Y 408.903,Z 301.461,A -85,B 0,C 180,E1 -11035.39,E2 -11035.39} C_VEL
LIN {X 0,Y 410.043,Z 220.966,A -85,B 0,C 180,E1 -11036.916,E2 -11036.916} C_VEL
LIN {X 0,Y 405.539,Z 208.228,A -85,B 0,C 180,E1 -11037.372,E2 -11037.372} C_VEL
LIN {X 0,Y 404.175,Z 204.142,A -85,B 0,C 180,E1 -11037.527,E2 -11037.527} C_VEL
LIN {X 0,Y 404.177,Z 204.141,A -85,B 0,C 180,E1 -11040.865,E2 -11040.865} C_VEL
LIN {X 0,Y 404.194,Z 204.14,A -85,B 0,C 180,E1 -11043.123,E2 -11043.123} C_VEL
LIN {X 0,Y 404.17,Z 204.14,A -85,B 0,C 180,E1 -11045.334,E2 -11045.334} C_VEL
LIN {X 0,Y 404.139,Z 204.142,A -85,B 0,C 180,E1 -11048.581,E2 -11048.581} C_VEL
LIN {X 0,Y 404.205,Z 204.132,A -85,B 0,C 180,E1 -11051.762,E2 -11051.762} C_VEL
LIN {X 0,Y 404.206,Z 204.138,A -85,B 0,C 180,E1 -11054.882,E2 -11054.882} C_VEL
LIN {X 0,Y 404.272,Z 204.13,A -85,B 0,C 180,E1 -11056.833,E2 -11056.833} C_VEL
LIN {X 0,Y 403.664,Z 204.201,A -85,B 0,C 180,E1 -11057.665,E2 -11057.665} C_VEL
LIN {X 0,Y 400.804,Z 204.559,A -85,B 0,C 180,E1 -11059.016,E2 -11059.016} C_VEL
LIN {X 0,Y 398.354,Z 204.866,A -85,B 0,C 180,E1 -11060.107,E2 -11060.107} C_VEL
LIN {X 0,Y 397.314,Z 204.994,A -85,B 0,C 180,E1 -11060.952,E2 -11060.952} C_VEL
LIN {X 0,Y 397.239,Z 205.001,A -85,B 0,C 180,E1 -11061.238,E2 -11061.238} C_VEL
LIN {X 0,Y 397.346,Z 204.986,A -85,B 0,C 180,E1 -11063.908,E2 -11063.908} C_VEL
LIN {X 0,Y 397.449,Z 204.974,A -85,B 0,C 180,E1 -11067.974,E2 -11067.974} C_VEL
LIN {X 0,Y 397.576,Z 204.959,A -85,B 0,C 180,E1 -11070,E2 -11070} C_VEL
LIN {X 0,Y 397.338,Z 204.988,A -85,B 0,C 180,E1 -11073.042,E2 -11073.042} C_VEL
LIN {X 0,Y 397.346,Z 204.99,A -85,B 0,C 180,E1 -11076.092,E2 -11076.092} C_VEL
LIN {X 0,Y 397.237,Z 205,A -85,B 0,C 180,E1 -11079.162,E2 -11079.162} C_VEL
LIN {X 0,Y 397.221,Z 205.008,A -85,B 0,C 180,E1 -11082.258,E2 -11082.258} C_VEL
LIN {X 0,Y 397.18,Z 205.007,A -85,B 0,C 180,E1 -11085.392,E2 -11085.392} C_VEL
LIN {X 0,Y 397.162,Z 205.011,A -85,B 0,C 180,E1 -11088.574,E2 -11088.574} C_VEL
LIN {X 0,Y 397.098,Z 205.022,A -85,B 0,C 180,E1 -11091.819,E2 -11091.819} C_VEL
LIN {X 0,Y 397.125,Z 205.014,A -85,B 0,C 180,E1 -11095.134,E2 -11095.134} C_VEL
LIN {X 0,Y 397.08,Z 205.02,A -85,B 0,C 180,E1 -11098.547,E2 -11098.547} C_VEL
LIN {X 0,Y 397.084,Z 205.025,A -85,B 0,C 180,E1 -11101.837,E2 -11101.837} C_VEL
LIN {X 0,Y 397.127,Z 205.014,A -85,B 0,C 180,E1 -11104.494,E2 -11104.494} C_VEL
LIN {X 0,Y 397.094,Z 205.018,A -85,B 0,C 180,E1 -11108.276,E2 -11108.276} C_VEL
LIN {X 0,Y 397.062,Z 205.022,A -85,B 0,C 180,E1 -11110.913,E2 -11110.913} C_VEL
LIN {X 0,Y 397.102,Z 205.021,A -85,B 0,C 180,E1 -11113.649,E2 -11113.649} C_VEL
LIN {X 0,Y 397.102,Z 205.016,A -85,B 0,C 180,E1 -11116.521,E2 -11116.521} C_VEL
LIN {X 0,Y 397.088,Z 205.018,A -85,B 0,C 180,E1 -11120.42,E2 -11120.42} C_VEL
LIN {X 0,Y 397.099,Z 205.021,A -85,B 0,C 180,E1 -11123.005,E2 -11123.005} C_VEL
LIN {X 0,Y 397.121,Z 205.014,A -85,B 0,C 180,E1 -11126.282,E2 -11126.282} C_VEL
LIN {X 0,Y 397.101,Z 205.016,A -85,B 0,C 180,E1 -11130.137,E2 -11130.137} C_VEL
LIN {X 0,Y 397.093,Z 205.018,A -85,B 0,C 180,E1 -11133.739,E2 -11133.739} C_VEL
LIN {X 0,Y 397.107,Z 205.021,A -85,B 0,C 180,E1 -11137.086,E2 -11137.086} C_VEL
LIN {X 0,Y 397.149,Z 205.012,A -85,B 0,C 180,E1 -11140.353,E2 -11140.353} C_VEL
LIN {X 0,Y 397.169,Z 205.008,A -85,B 0,C 180,E1 -11143.553,E2 -11143.553} C_VEL
LIN {X 0,Y 397.232,Z 205.007,A -85,B 0,C 180,E1 -11146.703,E2 -11146.703} C_VEL
LIN {X 0,Y 397.219,Z 205.002,A -85,B 0,C 180,E1 -11149.809,E2 -11149.809} C_VEL
LIN {X 0,Y 397.298,Z 204.995,A -85,B 0,C 180,E1 -11152.887,E2 -11152.887} C_VEL
LIN {X 0,Y 397.242,Z 205.001,A -85,B 0,C 180,E1 -11154.925,E2 -11154.925} C_VEL
LIN {X 0,Y 397.449,Z 204.975,A -85,B 0,C 180,E1 -11157.973,E2 -11157.973} C_VEL
LIN {X 0,Y 397.365,Z 204.984,A -85,B 0,C 180,E1 -11161.013,E2 -11161.013} C_VEL
LIN {X 0,Y 397.327,Z 204.989,A -85,B 0,C 180,E1 -11163.042,E2 -11163.042} C_VEL
LIN {X 0,Y 397.332,Z 204.993,A -85,B 0,C 180,E1 -11166.092,E2 -11166.092} C_VEL
LIN {X 0,Y 397.237,Z 205,A -85,B 0,C 180,E1 -11169.162,E2 -11169.162} C_VEL
LIN {X 0,Y 397.222,Z 205.006,A -85,B 0,C 180,E1 -11172.258,E2 -11172.258} C_VEL
LIN {X 0,Y 397.128,Z 205.014,A -85,B 0,C 180,E1 -11175.394,E2 -11175.394} C_VEL
LIN {X 0,Y 397.154,Z 205.011,A -85,B 0,C 180,E1 -11178.574,E2 -11178.574} C_VEL
LIN {X 0,Y 397.098,Z 205.024,A -85,B 0,C 180,E1 -11181.819,E2 -11181.819} C_VEL
LIN {X 0,Y 397.099,Z 205.018,A -85,B 0,C 180,E1 -11185.136,E2 -11185.136} C_VEL
LIN {X 0,Y 397.072,Z 205.02,A -85,B 0,C 180,E1 -11188.548,E2 -11188.548} C_VEL
LIN {X 0,Y 397.084,Z 205.023,A -85,B 0,C 180,E1 -11191.836,E2 -11191.836} C_VEL
LIN {X 0,Y 397.122,Z 205.014,A -85,B 0,C 180,E1 -11194.494,E2 -11194.494} C_VEL
LIN {X 0,Y 397.095,Z 205.018,A -85,B 0,C 180,E1 -11198.276,E2 -11198.276} C_VEL
LIN {X 0,Y 397.054,Z 205.023,A -85,B 0,C 180,E1 -11201.976,E2 -11201.976} C_VEL
LIN {X 0,Y 397.088,Z 205.023,A -85,B 0,C 180,E1 -11205.069,E2 -11205.069} C_VEL
LIN {X 0,Y 397.054,Z 205.023,A -85,B 0,C 180,E1 -11208.023,E2 -11208.023} C_VEL
LIN {X 0,Y 397.096,Z 205.018,A -85,B 0,C 180,E1 -11211.724,E2 -11211.724} C_VEL
LIN {X 0,Y 397.12,Z 205.018,A -85,B 0,C 180,E1 -11215.506,E2 -11215.506} C_VEL
LIN {X 0,Y 397.089,Z 205.024,A -85,B 0,C 180,E1 -11219.118,E2 -11219.118} C_VEL
LIN {X 0,Y 397.152,Z 205.152,A -85,B 0,C 180,E1 -11219.872,E2 -11219.872} C_VEL
LIN {X 0,Y 399.857,Z 218.015,A -85,B 0,C 180,E1 -11222.524,E2 -11222.524} C_VEL
LIN {X 0,Y 400.876,Z 224.455,A -85,B 0,C 180,E1 -11223.803,E2 -11223.803} C_VEL
LIN {X 0,Y 399.557,Z 243.045,A -85,B 0,C 180,E1 -11227.234,E2 -11227.234} C_VEL
LIN {X 0,Y 398.545,Z 259.243,A -85,B 0,C 180,E1 -11230.189,E2 -11230.189} C_VEL
LIN {X 0,Y 402.684,Z 292.844,A -85,B 0,C 180,E1 -11231.055,E2 -11231.055} C_VEL
LIN {X 0,Y 401.513,Z 369.212,A -85,B 0,C 180,E1 -11232.557,E2 -11232.557} C_VEL
LIN {X 0,Y 400.952,Z 382.676,A -85,B 0,C 180,E1 -11233.025,E2 -11233.025} C_VEL
LIN {X 0,Y 400.169,Z 395.493,A -85,B 0,C 180,E1 -11233.68,E2 -11233.68} C_VEL
LIN {X 0,Y 399.292,Z 408.055,A -85,B 0,C 180,E1 -11234.56,E2 -11234.56} C_VEL
LIN {X 0,Y 398.463,Z 419.313,A -85,B 0,C 180,E1 -11235.573,E2 -11235.573} C_VEL
LIN {X 0,Y 397.787,Z 429.465,A -85,B 0,C 180,E1 -11236.721,E2 -11236.721} C_VEL
LIN {X 0,Y 397.18,Z 438.657,A -85,B 0,C 180,E1 -11238,E2 -11238} C_VEL
LIN {X 0,Y 396.529,Z 447.615,A -85,B 0,C 180,E1 -11239.533,E2 -11239.533} C_VEL
LIN {X 0,Y 396.18,Z 454.778,A -85,B 0,C 180,E1 -11241.07,E2 -11241.07} C_VEL
LIN {X 0,Y 395.996,Z 461.312,A -85,B 0,C 180,E1 -11242.863,E2 -11242.863} C_VEL
LIN {X 0,Y 395.936,Z 465.589,A -85,B 0,C 180,E1 -11244.397,E2 -11244.397} C_VEL
LIN {X 0,Y 395.89,Z 468.754,A -85,B 0,C 180,E1 -11245.928,E2 -11245.928} C_VEL
LIN {X 0,Y 396.012,Z 470.324,A -85,B 0,C 180,E1 -11246.948,E2 -11246.948} C_VEL
LIN {X 0,Y 396.02,Z 471.422,A -85,B 0,C 180,E1 -11247.966,E2 -11247.966} C_VEL
LIN {X 0,Y 396.039,Z 472.088,A -85,B 0,C 180,E1 -11248.983,E2 -11248.983} C_VEL
LIN {X 0,Y 396.03,Z 472.347,A -85,B 0,C 180,E1 -11250,E2 -11250} C_VEL
LIN {X 0,Y 396.008,Z 472.201,A -85,B 0,C 180,E1 -11251.017,E2 -11251.017} C_VEL
LIN {X 0,Y 396.001,Z 471.606,A -85,B 0,C 180,E1 -11252.034,E2 -11252.034} C_VEL
LIN {X 0,Y 395.998,Z 470.591,A -85,B 0,C 180,E1 -11253.052,E2 -11253.052} C_VEL
LIN {X 0,Y 395.887,Z 469.16,A -85,B 0,C 180,E1 -11254.072,E2 -11254.072} C_VEL
LIN {X 0,Y 395.875,Z 466.178,A -85,B 0,C 180,E1 -11255.603,E2 -11255.603} C_VEL
LIN {X 0,Y 395.996,Z 462.144,A -85,B 0,C 180,E1 -11257.136,E2 -11257.136} C_VEL
LIN {X 0,Y 396.182,Z 455.973,A -85,B 0,C 180,E1 -11258.929,E2 -11258.929} C_VEL
LIN {X 0,Y 396.539,Z 449.202,A -85,B 0,C 180,E1 -11260.466,E2 -11260.466} C_VEL
LIN {X 0,Y 397.254,Z 440.828,A -85,B 0,C 180,E1 -11261.998,E2 -11261.998} C_VEL
LIN {X 0,Y 397.903,Z 432.3,A -85,B 0,C 180,E1 -11263.274,E2 -11263.274} C_VEL
LIN {X 0,Y 398.735,Z 421.868,A -85,B 0,C 180,E1 -11264.546,E2 -11264.546} C_VEL
LIN {X 0,Y 399.745,Z 410.14,A -85,B 0,C 180,E1 -11265.683,E2 -11265.683} C_VEL
LIN {X 0,Y 400.695,Z 398.647,A -85,B 0,C 180,E1 -11266.56,E2 -11266.56} C_VEL
LIN {X 0,Y 401.603,Z 385.656,A -85,B 0,C 180,E1 -11267.307,E2 -11267.307} C_VEL
LIN {X 0,Y 402.401,Z 371.951,A -85,B 0,C 180,E1 -11267.862,E2 -11267.862} C_VEL
LIN {X 0,Y 402.781,Z 359.706,A -85,B 0,C 180,E1 -11268.173,E2 -11268.173} C_VEL
LIN {X 0,Y 403.898,Z 291.728,A -85,B 0,C 180,E1 -11269.523,E2 -11269.523} C_VEL
LIN {X 0,Y 401.207,Z 270.285,A -85,B 0,C 180,E1 -11270.135,E2 -11270.135} C_VEL
LIN {X 0,Y 398.936,Z 256.1,A -85,B 0,C 180,E1 -11270.587,E2 -11270.587} C_VEL
LIN {X 0,Y 400.166,Z 236.756,A -85,B 0,C 180,E1 -11274.039,E2 -11274.039} C_VEL
LIN {X 0,Y 401.01,Z 223.51,A -85,B 0,C 180,E1 -11276.426,E2 -11276.426} C_VEL
LIN {X 0,Y 399.192,Z 213.786,A -85,B 0,C 180,E1 -11278.382,E2 -11278.382} C_VEL
LIN {X 0,Y 397.113,Z 205.024,A -85,B 0,C 180,E1 -11280.255,E2 -11280.255} C_VEL
LIN {X 0,Y 397.119,Z 205.018,A -85,B 0,C 180,E1 -11283.717,E2 -11283.717} C_VEL
LIN {X 0,Y 397.091,Z 205.021,A -85,B 0,C 180,E1 -11287.208,E2 -11287.208} C_VEL
LIN {X 0,Y 397.056,Z 205.027,A -85,B 0,C 180,E1 -11290.437,E2 -11290.437} C_VEL
LIN {X 0,Y 397.1,Z 205.017,A -85,B 0,C 180,E1 -11293.648,E2 -11293.648} C_VEL
LIN {X 0,Y 397.101,Z 205.021,A -85,B 0,C 180,E1 -11296.521,E2 -11296.521} C_VEL
LIN {X 0,Y 397.086,Z 205.022,A -85,B 0,C 180,E1 -11300.419,E2 -11300.419} C_VEL
LIN {X 0,Y 397.096,Z 205.02,A -85,B 0,C 180,E1 -11303.005,E2 -11303.005} C_VEL
LIN {X 0,Y 397.118,Z 205.021,A -85,B 0,C 180,E1 -11306.282,E2 -11306.282} C_VEL
LIN {X 0,Y 397.1,Z 205.019,A -85,B 0,C 180,E1 -11310.136,E2 -11310.136} C_VEL
LIN {X 0,Y 397.095,Z 205.017,A -85,B 0,C 180,E1 -11313.739,E2 -11313.739} C_VEL
LIN {X 0,Y 397.103,Z 205.016,A -85,B 0,C 180,E1 -11317.085,E2 -11317.085} C_VEL
LIN {X 0,Y 397.146,Z 205.015,A -85,B 0,C 180,E1 -11320.353,E2 -11320.353} C_VEL
LIN {X 0,Y 397.166,Z 205.01,A -85,B 0,C 180,E1 -11323.553,E2 -11323.553} C_VEL
LIN {X 0,Y 397.229,Z 205.002,A -85,B 0,C 180,E1 -11326.703,E2 -11326.703} C_VEL
LIN {X 0,Y 397.217,Z 205.007,A -85,B 0,C 180,E1 -11329.809,E2 -11329.809} C_VEL
LIN {X 0,Y 397.349,Z 204.989,A -85,B 0,C 180,E1 -11332.888,E2 -11332.888} C_VEL
LIN {X 0,Y 397.252,Z 205.001,A -85,B 0,C 180,E1 -11334.925,E2 -11334.925} C_VEL
LIN {X 0,Y 397.448,Z 204.975,A -85,B 0,C 180,E1 -11337.973,E2 -11337.973} C_VEL
LIN {X 0,Y 397.579,Z 204.96,A -85,B 0,C 180,E1 -11340,E2 -11340} C_VEL
LIN {X 0,Y 397.375,Z 204.987,A -85,B 0,C 180,E1 -11343.041,E2 -11343.041} C_VEL
LIN {X 0,Y 397.32,Z 204.991,A -85,B 0,C 180,E1 -11346.494,E2 -11346.494} C_VEL
LIN {X 0,Y 397.235,Z 205.006,A -85,B 0,C 180,E1 -11349.162,E2 -11349.162} C_VEL
LIN {X 0,Y 397.219,Z 205.01,A -85,B 0,C 180,E1 -11352.258,E2 -11352.258} C_VEL
LIN {X 0,Y 397.183,Z 205.016,A -85,B 0,C 180,E1 -11355.392,E2 -11355.392} C_VEL
LIN {X 0,Y 397.219,Z 205.182,A -85,B 0,C 180,E1 -11357.353,E2 -11357.353} C_VEL
LIN {X 0,Y 398.275,Z 207.944,A -85,B 0,C 180,E1 -11357.49,E2 -11357.49} C_VEL
LIN {X 0,Y 404.339,Z 222.541,A -85,B 0,C 180,E1 -11358.199,E2 -11358.199} C_VEL
LIN {X 0,Y 405.057,Z 224.442,A -85,B 0,C 180,E1 -11358.283,E2 -11358.283} C_VEL
LIN {X 0,Y 403.317,Z 312.857,A -85,B 0,C 180,E1 -11360.071,E2 -11360.071} C_VEL
LIN {X 0,Y 402.973,Z 325.387,A -85,B 0,C 180,E1 -11360.514,E2 -11360.514} C_VEL
LIN {X 0,Y 402.422,Z 338.319,A -85,B 0,C 180,E1 -11361.18,E2 -11361.18} C_VEL
LIN {X 0,Y 401.711,Z 349.973,A -85,B 0,C 180,E1 -11361.991,E2 -11361.991} C_VEL
LIN {X 0,Y 400.985,Z 360.738,A -85,B 0,C 180,E1 -11362.953,E2 -11362.953} C_VEL
LIN {X 0,Y 400.173,Z 370.609,A -85,B 0,C 180,E1 -11364.043,E2 -11364.043} C_VEL
LIN {X 0,Y 399.411,Z 379.591,A -85,B 0,C 180,E1 -11365.258,E2 -11365.258} C_VEL
LIN {X 0,Y 398.592,Z 388.323,A -85,B 0,C 180,E1 -11366.719,E2 -11366.719} C_VEL
LIN {X 0,Y 397.903,Z 395.422,A -85,B 0,C 180,E1 -11368.192,E2 -11368.192} C_VEL
LIN {X 0,Y 397.284,Z 401.983,A -85,B 0,C 180,E1 -11369.91,E2 -11369.91} C_VEL
LIN {X 0,Y 396.73,Z 407.249,A -85,B 0,C 180,E1 -11371.755,E2 -11371.755} C_VEL
LIN {X 0,Y 396.377,Z 410.896,A -85,B 0,C 180,E1 -11373.557,E2 -11373.557} C_VEL
LIN {X 0,Y 396.126,Z 413.136,A -85,B 0,C 180,E1 -11375.302,E2 -11375.302} C_VEL
LIN {X 0,Y 395.974,Z 414.165,A -85,B 0,C 180,E1 -11377.118,E2 -11377.118} C_VEL
LIN {X 0,Y 395.941,Z 414.043,A -85,B 0,C 180,E1 -11378.648,E2 -11378.648} C_VEL
LIN {X 0,Y 395.984,Z 412.921,A -85,B 0,C 180,E1 -11380.256,E2 -11380.256} C_VEL
LIN {X 0,Y 396.123,Z 410.832,A -85,B 0,C 180,E1 -11381.827,E2 -11381.827} C_VEL
LIN {X 0,Y 396.462,Z 406.867,A -85,B 0,C 180,E1 -11383.737,E2 -11383.737} C_VEL
LIN {X 0,Y 396.802,Z 402,A -85,B 0,C 180,E1 -11385.424,E2 -11385.424} C_VEL
LIN {X 0,Y 397.256,Z 395.485,A -85,B 0,C 180,E1 -11387.149,E2 -11387.149} C_VEL
LIN {X 0,Y 397.756,Z 388.634,A -85,B 0,C 180,E1 -11388.583,E2 -11388.583} C_VEL
LIN {X 0,Y 398.508,Z 379.282,A -85,B 0,C 180,E1 -11390.158,E2 -11390.158} C_VEL
LIN {X 0,Y 399.114,Z 370.863,A -85,B 0,C 180,E1 -11391.309,E2 -11391.309} C_VEL
LIN {X 0,Y 399.776,Z 360.258,A -85,B 0,C 180,E1 -11392.492,E2 -11392.492} C_VEL
LIN {X 0,Y 400.498,Z 349.06,A -85,B 0,C 180,E1 -11393.487,E2 -11393.487} C_VEL
LIN {X 0,Y 401.121,Z 337.54,A -85,B 0,C 180,E1 -11394.292,E2 -11394.292} C_VEL
LIN {X 0,Y 401.56,Z 324.646,A -85,B 0,C 180,E1 -11394.964,E2 -11394.964} C_VEL
LIN {X 0,Y 401.928,Z 311.301,A -85,B 0,C 180,E1 -11395.435,E2 -11395.435} C_VEL
LIN {X 0,Y 403.31,Z 222.614,A -85,B 0,C 180,E1 -11397.181,E2 -11397.181} C_VEL
LIN {X 0,Y 398.609,Z 209.343,A -85,B 0,C 180,E1 -11397.664,E2 -11397.664} C_VEL
LIN {X 0,Y 397.096,Z 205.023,A -85,B 0,C 180,E1 -11397.846,E2 -11397.846} C_VEL
LIN {X 0,Y 397.122,Z 205.018,A -85,B 0,C 180,E1 -11401.457,E2 -11401.457} C_VEL
LIN {X 0,Y 397.151,Z 205.011,A -85,B 0,C 180,E1 -11404.489,E2 -11404.489} C_VEL
LIN {X 0,Y 397.096,Z 205.017,A -85,B 0,C 180,E1 -11408.182,E2 -11408.182} C_VEL
LIN {X 0,Y 397.158,Z 205.011,A -85,B 0,C 180,E1 -11411.427,E2 -11411.427} C_VEL
LIN {X 0,Y 397.179,Z 205.011,A -85,B 0,C 180,E1 -11414.608,E2 -11414.608} C_VEL
LIN {X 0,Y 397.22,Z 205.002,A -85,B 0,C 180,E1 -11417.742,E2 -11417.742} C_VEL
LIN {X 0,Y 397.239,Z 205.001,A -85,B 0,C 180,E1 -11421.238,E2 -11421.238} C_VEL
LIN {X 0,Y 396.595,Z 205.082,A -85,B 0,C 180,E1 -11422.085,E2 -11422.085} C_VEL
LIN {X 0,Y 393.738,Z 205.436,A -85,B 0,C 180,E1 -11423.461,E2 -11423.461} C_VEL
LIN {X 0,Y 391.288,Z 205.747,A -85,B 0,C 180,E1 -11424.572,E2 -11424.572} C_VEL
LIN {X 0,Y 390.211,Z 205.876,A -85,B 0,C 180,E1 -11425.432,E2 -11425.432} C_VEL
LIN {X 0,Y 390.111,Z 205.887,A -85,B 0,C 180,E1 -11425.724,E2 -11425.724} C_VEL
LIN {X 0,Y 390.417,Z 205.85,A -85,B 0,C 180,E1 -11427.937,E2 -11427.937} C_VEL
LIN {X 0,Y 390.545,Z 205.835,A -85,B 0,C 180,E1 -11430,E2 -11430} C_VEL
LIN {X 0,Y 390.274,Z 205.868,A -85,B 0,C 180,E1 -11433.097,E2 -11433.097} C_VEL
LIN {X 0,Y 390.3,Z 205.869,A -85,B 0,C 180,E1 -11436.203,E2 -11436.203} C_VEL
LIN {X 0,Y 390.195,Z 205.877,A -85,B 0,C 180,E1 -11439.329,E2 -11439.329} C_VEL
LIN {X 0,Y 390.172,Z 205.883,A -85,B 0,C 180,E1 -11442.483,E2 -11442.483} C_VEL
LIN {X 0,Y 390.14,Z 205.886,A -85,B 0,C 180,E1 -11445.677,E2 -11445.677} C_VEL
LIN {X 0,Y 390.106,Z 205.888,A -85,B 0,C 180,E1 -11448.922,E2 -11448.922} C_VEL
LIN {X 0,Y 390.039,Z 205.9,A -85,B 0,C 180,E1 -11452.235,E2 -11452.235} C_VEL
LIN {X 0,Y 390.086,Z 205.895,A -85,B 0,C 180,E1 -11455.733,E2 -11455.733} C_VEL
LIN {X 0,Y 390.035,Z 205.897,A -85,B 0,C 180,E1 -11459.112,E2 -11459.112} C_VEL
LIN {X 0,Y 390.045,Z 205.896,A -85,B 0,C 180,E1 -11462.722,E2 -11462.722} C_VEL
LIN {X 0,Y 390.057,Z 205.899,A -85,B 0,C 180,E1 -11465.825,E2 -11465.825} C_VEL
LIN {X 0,Y 390.039,Z 205.899,A -85,B 0,C 180,E1 -11469.213,E2 -11469.213} C_VEL
LIN {X 0,Y 390.039,Z 205.896,A -85,B 0,C 180,E1 -11472.373,E2 -11472.373} C_VEL
LIN {X 0,Y 390.046,Z 205.902,A -85,B 0,C 180,E1 -11475.355,E2 -11475.355} C_VEL
LIN {X 0,Y 390.022,Z 205.899,A -85,B 0,C 180,E1 -11478.185,E2 -11478.185} C_VEL
LIN {X 0,Y 390.06,Z 205.896,A -85,B 0,C 180,E1 -11480.904,E2 -11480.904} C_VEL
LIN {X 0,Y 390.087,Z 205.893,A -85,B 0,C 180,E1 -11484.793,E2 -11484.793} C_VEL
LIN {X 0,Y 390.025,Z 205.899,A -85,B 0,C 180,E1 -11488.496,E2 -11488.496} C_VEL
LIN {X 0,Y 390.032,Z 205.897,A -85,B 0,C 180,E1 -11492.063,E2 -11492.063} C_VEL
LIN {X 0,Y 390.056,Z 205.895,A -85,B 0,C 180,E1 -11495.518,E2 -11495.518} C_VEL
LIN {X 0,Y 390.058,Z 205.901,A -85,B 0,C 180,E1 -11498.878,E2 -11498.878} C_VEL
LIN {X 0,Y 390.114,Z 205.888,A -85,B 0,C 180,E1 -11502.166,E2 -11502.166} C_VEL
LIN {X 0,Y 390.146,Z 205.884,A -85,B 0,C 180,E1 -11505.393,E2 -11505.393} C_VEL
LIN {X 0,Y 390.15,Z 205.889,A -85,B 0,C 180,E1 -11508.571,E2 -11508.571} C_VEL
LIN {X 0,Y 390.26,Z 205.871,A -85,B 0,C 180,E1 -11512.086,E2 -11512.086} C_VEL
LIN {X 0,Y 390.213,Z 205.878,A -85,B 0,C 180,E1 -11514.833,E2 -11514.833} C_VEL
LIN {X 0,Y 390.417,Z 205.851,A -85,B 0,C 180,E1 -11517.937,E2 -11517.937} C_VEL
LIN {X 0,Y 390.331,Z 205.861,A -85,B 0,C 180,E1 -11521.032,E2 -11521.032} C_VEL
LIN {X 0,Y 390.263,Z 205.869,A -85,B 0,C 180,E1 -11523.097,E2 -11523.097} C_VEL
LIN {X 0,Y 390.286,Z 205.872,A -85,B 0,C 180,E1 -11526.203,E2 -11526.203} C_VEL
LIN {X 0,Y 390.195,Z 205.877,A -85,B 0,C 180,E1 -11529.329,E2 -11529.329} C_VEL
LIN {X 0,Y 390.174,Z 205.882,A -85,B 0,C 180,E1 -11532.483,E2 -11532.483} C_VEL
LIN {X 0,Y 390.071,Z 205.896,A -85,B 0,C 180,E1 -11535.68,E2 -11535.68} C_VEL
LIN {X 0,Y 390.101,Z 205.889,A -85,B 0,C 180,E1 -11538.922,E2 -11538.922} C_VEL
LIN {X 0,Y 390.038,Z 205.899,A -85,B 0,C 180,E1 -11542.234,E2 -11542.234} C_VEL
LIN {X 0,Y 390.052,Z 205.901,A -85,B 0,C 180,E1 -11545.722,E2 -11545.722} C_VEL
LIN {X 0,Y 390.031,Z 205.899,A -85,B 0,C 180,E1 -11549.112,E2 -11549.112} C_VEL
LIN {X 0,Y 390.044,Z 205.896,A -85,B 0,C 180,E1 -11552.722,E2 -11552.722} C_VEL
LIN {X 0,Y 390.056,Z 205.897,A -85,B 0,C 180,E1 -11555.825,E2 -11555.825} C_VEL
LIN {X 0,Y 390.04,Z 205.9,A -85,B 0,C 180,E1 -11559.212,E2 -11559.212} C_VEL
LIN {X 0,Y 390.032,Z 205.897,A -85,B 0,C 180,E1 -11562.372,E2 -11562.372} C_VEL
LIN {X 0,Y 390.043,Z 205.902,A -85,B 0,C 180,E1 -11565.354,E2 -11565.354} C_VEL
LIN {X 0,Y 390.017,Z 205.899,A -85,B 0,C 180,E1 -11568.184,E2 -11568.184} C_VEL
LIN {X 0,Y 390.062,Z 205.897,A -85,B 0,C 180,E1 -11570.904,E2 -11570.904} C_VEL
LIN {X 0,Y 390.072,Z 205.896,A -85,B 0,C 180,E1 -11574.791,E2 -11574.791} C_VEL
LIN {X 0,Y 390.028,Z 205.902,A -85,B 0,C 180,E1 -11578.496,E2 -11578.496} C_VEL
LIN {X 0,Y 390.091,Z 205.961,A -85,B 0,C 180,E1 -11579.592,E2 -11579.592} C_VEL
LIN {X 0,Y 393.045,Z 220.057,A -85,B 0,C 180,E1 -11582.552,E2 -11582.552} C_VEL
LIN {X 0,Y 393.925,Z 226.247,A -85,B 0,C 180,E1 -11583.796,E2 -11583.796} C_VEL
LIN {X 0,Y 392.481,Z 245.244,A -85,B 0,C 180,E1 -11587.356,E2 -11587.356} C_VEL
LIN {X 0,Y 391.589,Z 258.784,A -85,B 0,C 180,E1 -11589.874,E2 -11589.874} C_VEL
LIN {X 0,Y 395.864,Z 293.023,A -85,B 0,C 180,E1 -11590.776,E2 -11590.776} C_VEL
LIN {X 0,Y 394.649,Z 369.1,A -85,B 0,C 180,E1 -11592.311,E2 -11592.311} C_VEL
LIN {X 0,Y 394.058,Z 382.425,A -85,B 0,C 180,E1 -11592.785,E2 -11592.785} C_VEL
LIN {X 0,Y 393.257,Z 395.157,A -85,B 0,C 180,E1 -11593.451,E2 -11593.451} C_VEL
LIN {X 0,Y 392.44,Z 406.899,A -85,B 0,C 180,E1 -11594.284,E2 -11594.284} C_VEL
LIN {X 0,Y 391.537,Z 418.275,A -85,B 0,C 180,E1 -11595.313,E2 -11595.313} C_VEL
LIN {X 0,Y 390.82,Z 428.564,A -85,B 0,C 180,E1 -11596.48,E2 -11596.48} C_VEL
LIN {X 0,Y 390.138,Z 437.823,A -85,B 0,C 180,E1 -11597.78,E2 -11597.78} C_VEL
LIN {X 0,Y 389.513,Z 446.849,A -85,B 0,C 180,E1 -11599.342,E2 -11599.342} C_VEL
LIN {X 0,Y 389.123,Z 454.081,A -85,B 0,C 180,E1 -11600.907,E2 -11600.907} C_VEL
LIN {X 0,Y 388.922,Z 460.657,A -85,B 0,C 180,E1 -11602.733,E2 -11602.733} C_VEL
LIN {X 0,Y 388.837,Z 464.489,A -85,B 0,C 180,E1 -11604.098,E2 -11604.098} C_VEL
LIN {X 0,Y 388.81,Z 468.162,A -85,B 0,C 180,E1 -11605.853,E2 -11605.853} C_VEL
LIN {X 0,Y 388.927,Z 469.745,A -85,B 0,C 180,E1 -11606.892,E2 -11606.892} C_VEL
LIN {X 0,Y 388.948,Z 470.868,A -85,B 0,C 180,E1 -11607.929,E2 -11607.929} C_VEL
LIN {X 0,Y 388.957,Z 471.544,A -85,B 0,C 180,E1 -11608.964,E2 -11608.964} C_VEL
LIN {X 0,Y 388.978,Z 471.816,A -85,B 0,C 180,E1 -11610,E2 -11610} C_VEL
LIN {X 0,Y 388.927,Z 471.679,A -85,B 0,C 180,E1 -11611.035,E2 -11611.035} C_VEL
LIN {X 0,Y 388.93,Z 471.106,A -85,B 0,C 180,E1 -11612.071,E2 -11612.071} C_VEL
LIN {X 0,Y 388.898,Z 470.1,A -85,B 0,C 180,E1 -11613.108,E2 -11613.108} C_VEL
LIN {X 0,Y 388.803,Z 468.68,A -85,B 0,C 180,E1 -11614.146,E2 -11614.146} C_VEL
LIN {X 0,Y 388.781,Z 465.447,A -85,B 0,C 180,E1 -11615.829,E2 -11615.829} C_VEL
LIN {X 0,Y 388.922,Z 461.701,A -85,B 0,C 180,E1 -11617.267,E2 -11617.267} C_VEL
LIN {X 0,Y 389.124,Z 455.561,A -85,B 0,C 180,E1 -11619.093,E2 -11619.093} C_VEL
LIN {X 0,Y 389.533,Z 448.815,A -85,B 0,C 180,E1 -11620.657,E2 -11620.657} C_VEL
LIN {X 0,Y 390.282,Z 440.464,A -85,B 0,C 180,E1 -11622.215,E2 -11622.215} C_VEL
LIN {X 0,Y 391.038,Z 430.912,A -85,B 0,C 180,E1 -11623.664,E2 -11623.664} C_VEL
LIN {X 0,Y 391.947,Z 420.449,A -85,B 0,C 180,E1 -11624.937,E2 -11624.937} C_VEL
LIN {X 0,Y 393.057,Z 408.577,A -85,B 0,C 180,E1 -11626.09,E2 -11626.09} C_VEL
LIN {X 0,Y 393.996,Z 396.783,A -85,B 0,C 180,E1 -11626.983,E2 -11626.983} C_VEL
LIN {X 0,Y 395.059,Z 383.386,A -85,B 0,C 180,E1 -11627.737,E2 -11627.737} C_VEL
LIN {X 0,Y 395.815,Z 370.775,A -85,B 0,C 180,E1 -11628.237,E2 -11628.237} C_VEL
LIN {X 0,Y 396.23,Z 354.92,A -85,B 0,C 180,E1 -11628.618,E2 -11628.618} C_VEL
LIN {X 0,Y 397.275,Z 292.063,A -85,B 0,C 180,E1 -11629.898,E2 -11629.898} C_VEL
LIN {X 0,Y 394.701,Z 271.561,A -85,B 0,C 180,E1 -11630.501,E2 -11630.501} C_VEL
LIN {X 0,Y 392.119,Z 255.369,A -85,B 0,C 180,E1 -11631.052,E2 -11631.052} C_VEL
LIN {X 0,Y 393.539,Z 234.65,A -85,B 0,C 180,E1 -11634.813,E2 -11634.813} C_VEL
LIN {X 0,Y 394.132,Z 224.604,A -85,B 0,C 180,E1 -11636.677,E2 -11636.677} C_VEL
LIN {X 0,Y 391.931,Z 213.575,A -85,B 0,C 180,E1 -11638.957,E2 -11638.957} C_VEL
LIN {X 0,Y 390.047,Z 205.903,A -85,B 0,C 180,E1 -11640.673,E2 -11640.673} C_VEL
LIN {X 0,Y 390.069,Z 205.897,A -85,B 0,C 180,E1 -11644.024,E2 -11644.024} C_VEL
LIN {X 0,Y 390.04,Z 205.899,A -85,B 0,C 180,E1 -11647.55,E2 -11647.55} C_VEL
LIN {X 0,Y 390.019,Z 205.901,A -85,B 0,C 180,E1 -11650.815,E2 -11650.815} C_VEL
LIN {X 0,Y 390.054,Z 205.896,A -85,B 0,C 180,E1 -11653.886,E2 -11653.886} C_VEL
LIN {X 0,Y 390.055,Z 205.896,A -85,B 0,C 180,E1 -11656.789,E2 -11656.789} C_VEL
LIN {X 0,Y 390.011,Z 205.9,A -85,B 0,C 180,E1 -11659.555,E2 -11659.555} C_VEL
LIN {X 0,Y 390.039,Z 205.899,A -85,B 0,C 180,E1 -11662.45,E2 -11662.45} C_VEL
LIN {X 0,Y 390.068,Z 205.895,A -85,B 0,C 180,E1 -11665.975,E2 -11665.975} C_VEL
LIN {X 0,Y 390.037,Z 205.9,A -85,B 0,C 180,E1 -11669.7,E2 -11669.7} C_VEL
LIN {X 0,Y 390.055,Z 205.893,A -85,B 0,C 180,E1 -11673.227,E2 -11673.227} C_VEL
LIN {X 0,Y 390.067,Z 205.893,A -85,B 0,C 180,E1 -11676.764,E2 -11676.764} C_VEL
LIN {X 0,Y 390.103,Z 205.89,A -85,B 0,C 180,E1 -11679.983,E2 -11679.983} C_VEL
LIN {X 0,Y 390.138,Z 205.883,A -85,B 0,C 180,E1 -11683.248,E2 -11683.248} C_VEL
LIN {X 0,Y 390.194,Z 205.878,A -85,B 0,C 180,E1 -11686.561,E2 -11686.561} C_VEL
LIN {X 0,Y 390.205,Z 205.876,A -85,B 0,C 180,E1 -11690.671,E2 -11690.671} C_VEL
LIN {X 0,Y 390.324,Z 205.863,A -85,B 0,C 180,E1 -11693.798,E2 -11693.798} C_VEL
LIN {X 0,Y 390.417,Z 205.851,A -85,B 0,C 180,E1 -11697.937,E2 -11697.937} C_VEL
LIN {X 0,Y 390.548,Z 205.836,A -85,B 0,C 180,E1 -11700,E2 -11700} C_VEL
LIN {X 0,Y 390.31,Z 205.867,A -85,B 0,C 180,E1 -11703.096,E2 -11703.096} C_VEL
LIN {X 0,Y 390.278,Z 205.868,A -85,B 0,C 180,E1 -11706.485,E2 -11706.485} C_VEL
LIN {X 0,Y 390.193,Z 205.883,A -85,B 0,C 180,E1 -11709.329,E2 -11709.329} C_VEL
LIN {X 0,Y 390.171,Z 205.889,A -85,B 0,C 180,E1 -11712.483,E2 -11712.483} C_VEL
LIN {X 0,Y 390.147,Z 205.891,A -85,B 0,C 180,E1 -11715.676,E2 -11715.676} C_VEL
LIN {X 0,Y 390.168,Z 205.888,A -85,B 0,C 180,E1 -11716.878,E2 -11716.878} C_VEL
LIN {X 0,Y 391.299,Z 208.912,A -85,B 0,C 180,E1 -11717.04,E2 -11717.04} C_VEL
LIN {X 0,Y 397.319,Z 222.917,A -85,B 0,C 180,E1 -11717.761,E2 -11717.761} C_VEL
LIN {X 0,Y 398.492,Z 226.215,A -85,B 0,C 180,E1 -11717.911,E2 -11717.911} C_VEL
LIN {X 0,Y 396.703,Z 313.403,A -85,B 0,C 180,E1 -11719.717,E2 -11719.717} C_VEL
LIN {X 0,Y 396.337,Z 326.009,A -85,B 0,C 180,E1 -11720.171,E2 -11720.171} C_VEL
LIN {X 0,Y 395.776,Z 338.182,A -85,B 0,C 180,E1 -11720.803,E2 -11720.803} C_VEL
LIN {X 0,Y 395.006,Z 350.496,A -85,B 0,C 180,E1 -11721.665,E2 -11721.665} C_VEL
LIN {X 0,Y 394.187,Z 361.88,A -85,B 0,C 180,E1 -11722.704,E2 -11722.704} C_VEL
LIN {X 0,Y 393.329,Z 371.824,A -85,B 0,C 180,E1 -11723.833,E2 -11723.833} C_VEL
LIN {X 0,Y 392.458,Z 381.306,A -85,B 0,C 180,E1 -11725.17,E2 -11725.17} C_VEL
LIN {X 0,Y 391.596,Z 389.816,A -85,B 0,C 180,E1 -11726.659,E2 -11726.659} C_VEL
LIN {X 0,Y 390.852,Z 397.03,A -85,B 0,C 180,E1 -11728.227,E2 -11728.227} C_VEL
LIN {X 0,Y 390.363,Z 402.129,A -85,B 0,C 180,E1 -11729.612,E2 -11729.612} C_VEL
LIN {X 0,Y 389.733,Z 407.621,A -85,B 0,C 180,E1 -11731.531,E2 -11731.531} C_VEL
LIN {X 0,Y 389.474,Z 410.296,A -85,B 0,C 180,E1 -11732.775,E2 -11732.775} C_VEL
LIN {X 0,Y 389.229,Z 412.322,A -85,B 0,C 180,E1 -11734.038,E2 -11734.038} C_VEL
LIN {X 0,Y 389.021,Z 413.989,A -85,B 0,C 180,E1 -11735.614,E2 -11735.614} C_VEL
LIN {X 0,Y 388.878,Z 414.725,A -85,B 0,C 180,E1 -11737.327,E2 -11737.327} C_VEL
LIN {X 0,Y 388.874,Z 414.248,A -85,B 0,C 180,E1 -11739.238,E2 -11739.238} C_VEL
LIN {X 0,Y 388.936,Z 413.017,A -85,B 0,C 180,E1 -11740.63,E2 -11740.63} C_VEL
LIN {X 0,Y 389.111,Z 410.694,A -85,B 0,C 180,E1 -11742.224,E2 -11742.224} C_VEL
LIN {X 0,Y 389.418,Z 407.394,A -85,B 0,C 180,E1 -11743.789,E2 -11743.789} C_VEL
LIN {X 0,Y 389.794,Z 401.958,A -85,B 0,C 180,E1 -11745.683,E2 -11745.683} C_VEL
LIN {X 0,Y 390.192,Z 396.509,A -85,B 0,C 180,E1 -11747.143,E2 -11747.143} C_VEL
LIN {X 0,Y 390.7,Z 389.771,A -85,B 0,C 180,E1 -11748.604,E2 -11748.604} C_VEL
LIN {X 0,Y 391.43,Z 380.902,A -85,B 0,C 180,E1 -11750.15,E2 -11750.15} C_VEL
LIN {X 0,Y 392.073,Z 372.361,A -85,B 0,C 180,E1 -11751.366,E2 -11751.366} C_VEL
LIN {X 0,Y 392.74,Z 362.465,A -85,B 0,C 180,E1 -11752.525,E2 -11752.525} C_VEL
LIN {X 0,Y 393.493,Z 351.118,A -85,B 0,C 180,E1 -11753.584,E2 -11753.584} C_VEL
LIN {X 0,Y 394.219,Z 339.142,A -85,B 0,C 180,E1 -11754.456,E2 -11754.456} C_VEL
LIN {X 0,Y 394.713,Z 326.88,A -85,B 0,C 180,E1 -11755.134,E2 -11755.134} C_VEL
LIN {X 0,Y 395.016,Z 314.085,A -85,B 0,C 180,E1 -11755.626,E2 -11755.626} C_VEL
LIN {X 0,Y 395.318,Z 296.522,A -85,B 0,C 180,E1 -11756.021,E2 -11756.021} C_VEL
LIN {X 0,Y 396.474,Z 223.74,A -85,B 0,C 180,E1 -11757.464,E2 -11757.464} C_VEL
LIN {X 0,Y 390.075,Z 205.963,A -85,B 0,C 180,E1 -11758.137,E2 -11758.137} C_VEL
LIN {X 0,Y 390.118,Z 205.887,A -85,B 0,C 180,E1 -11762.07,E2 -11762.07} C_VEL
LIN {X 0,Y 390.075,Z 205.894,A -85,B 0,C 180,E1 -11765.519,E2 -11765.519} C_VEL
LIN {X 0,Y 390.088,Z 205.892,A -85,B 0,C 180,E1 -11769.53,E2 -11769.53} C_VEL
LIN {X 0,Y 390.139,Z 205.887,A -85,B 0,C 180,E1 -11773.249,E2 -11773.249} C_VEL
LIN {X 0,Y 390.195,Z 205.881,A -85,B 0,C 180,E1 -11776.562,E2 -11776.562} C_VEL
LIN {X 0,Y 390.168,Z 205.88,A -85,B 0,C 180,E1 -11779.623,E2 -11779.623} C_VEL
LIN {X 0,Y 390.269,Z 205.874,A -85,B 0,C 180,E1 -11782.758,E2 -11782.758} C_VEL
LIN {X 0,Y 390.218,Z 205.878,A -85,B 0,C 180,E1 -11784.834,E2 -11784.834} C_VEL
LIN {X 0,Y 390.111,Z 205.887,A -85,B 0,C 180,E1 -11785.724,E2 -11785.724} C_VEL
LIN {X 0,Y 389.48,Z 205.973,A -85,B 0,C 180,E1 -11786.586,E2 -11786.586} C_VEL
LIN {X 0,Y 386.877,Z 206.294,A -85,B 0,C 180,E1 -11787.994,E2 -11787.994} C_VEL
LIN {X 0,Y 383.831,Z 206.672,A -85,B 0,C 180,E1 -11789.71,E2 -11789.71} C_VEL
LIN {X 0,Y 383.443,Z 206.718,A -85,B 0,C 180,E1 -11790.3,E2 -11790.3} C_VEL
LIN {X 0,Y 383.212,Z 206.747,A -85,B 0,C 180,E1 -11793.154,E2 -11793.154} C_VEL
LIN {X 0,Y 383.257,Z 206.748,A -85,B 0,C 180,E1 -11796.317,E2 -11796.317} C_VEL
LIN {X 0,Y 383.145,Z 206.755,A -85,B 0,C 180,E1 -11799.503,E2 -11799.503} C_VEL
LIN {X 0,Y 383.127,Z 206.758,A -85,B 0,C 180,E1 -11803.536,E2 -11803.536} C_VEL
LIN {X 0,Y 383.096,Z 206.762,A -85,B 0,C 180,E1 -11807.455,E2 -11807.455} C_VEL
LIN {X 0,Y 383.031,Z 206.77,A -85,B 0,C 180,E1 -11810.647,E2 -11810.647} C_VEL
LIN {X 0,Y 383.018,Z 206.776,A -85,B 0,C 180,E1 -11813.809,E2 -11813.809} C_VEL
LIN {X 0,Y 382.995,Z 206.775,A -85,B 0,C 180,E1 -11817.307,E2 -11817.307} C_VEL
LIN {X 0,Y 382.984,Z 206.775,A -85,B 0,C 180,E1 -11820.919,E2 -11820.919} C_VEL
LIN {X 0,Y 383.02,Z 206.771,A -85,B 0,C 180,E1 -11824.668,E2 -11824.668} C_VEL
LIN {X 0,Y 382.995,Z 206.777,A -85,B 0,C 180,E1 -11827.903,E2 -11827.903} C_VEL
LIN {X 0,Y 382.969,Z 206.782,A -85,B 0,C 180,E1 -11831.35,E2 -11831.35} C_VEL
LIN {X 0,Y 382.997,Z 206.774,A -85,B 0,C 180,E1 -11834.303,E2 -11834.303} C_VEL
LIN {X 0,Y 383.012,Z 206.777,A -85,B 0,C 180,E1 -11837.24,E2 -11837.24} C_VEL
LIN {X 0,Y 382.988,Z 206.775,A -85,B 0,C 180,E1 -11840.419,E2 -11840.419} C_VEL
LIN {X 0,Y 383.026,Z 206.77,A -85,B 0,C 180,E1 -11844.045,E2 -11844.045} C_VEL
LIN {X 0,Y 382.989,Z 206.777,A -85,B 0,C 180,E1 -11847.578,E2 -11847.578} C_VEL
LIN {X 0,Y 382.98,Z 206.776,A -85,B 0,C 180,E1 -11850.299,E2 -11850.299} C_VEL
LIN {X 0,Y 383.006,Z 206.772,A -85,B 0,C 180,E1 -11854.045,E2 -11854.045} C_VEL
LIN {X 0,Y 382.994,Z 206.776,A -85,B 0,C 180,E1 -11857.334,E2 -11857.334} C_VEL
LIN {X 0,Y 383.061,Z 206.771,A -85,B 0,C 180,E1 -11860.716,E2 -11860.716} C_VEL
LIN {X 0,Y 383.083,Z 206.763,A -85,B 0,C 180,E1 -11864.027,E2 -11864.027} C_VEL
LIN {X 0,Y 383.139,Z 206.757,A -85,B 0,C 180,E1 -11867.284,E2 -11867.284} C_VEL
LIN {X 0,Y 383.146,Z 206.761,A -85,B 0,C 180,E1 -11870.498,E2 -11870.498} C_VEL
LIN {X 0,Y 383.245,Z 206.743,A -85,B 0,C 180,E1 -11873.683,E2 -11873.683} C_VEL
LIN {X 0,Y 383.383,Z 206.727,A -85,B 0,C 180,E1 -11877.899,E2 -11877.899} C_VEL
LIN {X 0,Y 383.299,Z 206.737,A -85,B 0,C 180,E1 -11881.051,E2 -11881.051} C_VEL
LIN {X 0,Y 383.201,Z 206.748,A -85,B 0,C 180,E1 -11883.154,E2 -11883.154} C_VEL
LIN {X 0,Y 383.242,Z 206.749,A -85,B 0,C 180,E1 -11886.317,E2 -11886.317} C_VEL
LIN {X 0,Y 383.145,Z 206.756,A -85,B 0,C 180,E1 -11889.502,E2 -11889.502} C_VEL
LIN {X 0,Y 383.129,Z 206.759,A -85,B 0,C 180,E1 -11893.536,E2 -11893.536} C_VEL
LIN {X 0,Y 383.061,Z 206.767,A -85,B 0,C 180,E1 -11897.437,E2 -11897.437} C_VEL
LIN {X 0,Y 383.032,Z 206.77,A -85,B 0,C 180,E1 -11900.647,E2 -11900.647} C_VEL
LIN {X 0,Y 383.013,Z 206.778,A -85,B 0,C 180,E1 -11903.809,E2 -11903.809} C_VEL
LIN {X 0,Y 382.984,Z 206.778,A -85,B 0,C 180,E1 -11907.308,E2 -11907.308} C_VEL
LIN {X 0,Y 382.984,Z 206.776,A -85,B 0,C 180,E1 -11910.919,E2 -11910.919} C_VEL
LIN {X 0,Y 383.019,Z 206.771,A -85,B 0,C 180,E1 -11914.668,E2 -11914.668} C_VEL
LIN {X 0,Y 382.996,Z 206.776,A -85,B 0,C 180,E1 -11917.902,E2 -11917.902} C_VEL
LIN {X 0,Y 382.963,Z 206.784,A -85,B 0,C 180,E1 -11921.35,E2 -11921.35} C_VEL
LIN {X 0,Y 382.991,Z 206.774,A -85,B 0,C 180,E1 -11924.302,E2 -11924.302} C_VEL
LIN {X 0,Y 383.013,Z 206.778,A -85,B 0,C 180,E1 -11927.24,E2 -11927.24} C_VEL
LIN {X 0,Y 382.989,Z 206.775,A -85,B 0,C 180,E1 -11930.419,E2 -11930.419} C_VEL
LIN {X 0,Y 383.017,Z 206.771,A -85,B 0,C 180,E1 -11934.043,E2 -11934.043} C_VEL
LIN {X 0,Y 382.987,Z 206.778,A -85,B 0,C 180,E1 -11937.578,E2 -11937.578} C_VEL
LIN {X 0,Y 383.056,Z 206.948,A -85,B 0,C 180,E1 -11939.346,E2 -11939.346} C_VEL
LIN {X 0,Y 385.711,Z 219.403,A -85,B 0,C 180,E1 -11942.018,E2 -11942.018} C_VEL
LIN {X 0,Y 386.979,Z 226.961,A -85,B 0,C 180,E1 -11943.58,E2 -11943.58} C_VEL
LIN {X 0,Y 385.49,Z 245.945,A -85,B 0,C 180,E1 -11947.206,E2 -11947.206} C_VEL
LIN {X 0,Y 384.665,Z 258.317,A -85,B 0,C 180,E1 -11949.548,E2 -11949.548} C_VEL
LIN {X 0,Y 389.037,Z 293.513,A -85,B 0,C 180,E1 -11950.498,E2 -11950.498} C_VEL
LIN {X 0,Y 387.8,Z 367.866,A -85,B 0,C 180,E1 -11952.022,E2 -11952.022} C_VEL
LIN {X 0,Y 387.178,Z 381.406,A -85,B 0,C 180,E1 -11952.504,E2 -11952.504} C_VEL
LIN {X 0,Y 386.411,Z 393.784,A -85,B 0,C 180,E1 -11953.15,E2 -11953.15} C_VEL
LIN {X 0,Y 385.585,Z 405.727,A -85,B 0,C 180,E1 -11953.997,E2 -11953.997} C_VEL
LIN {X 0,Y 384.596,Z 417.215,A -85,B 0,C 180,E1 -11955.041,E2 -11955.041} C_VEL
LIN {X 0,Y 383.838,Z 427.626,A -85,B 0,C 180,E1 -11956.23,E2 -11956.23} C_VEL
LIN {X 0,Y 383.106,Z 436.965,A -85,B 0,C 180,E1 -11957.552,E2 -11957.552} C_VEL
LIN {X 0,Y 382.581,Z 444.673,A -85,B 0,C 180,E1 -11958.879,E2 -11958.879} C_VEL
LIN {X 0,Y 382.113,Z 452.223,A -85,B 0,C 180,E1 -11960.472,E2 -11960.472} C_VEL
LIN {X 0,Y 381.879,Z 458.273,A -85,B 0,C 180,E1 -11962.066,E2 -11962.066} C_VEL
LIN {X 0,Y 381.806,Z 463.188,A -85,B 0,C 180,E1 -11963.718,E2 -11963.718} C_VEL
LIN {X 0,Y 381.778,Z 466.618,A -85,B 0,C 180,E1 -11965.248,E2 -11965.248} C_VEL
LIN {X 0,Y 381.83,Z 469.154,A -85,B 0,C 180,E1 -11966.834,E2 -11966.834} C_VEL
LIN {X 0,Y 381.877,Z 470.308,A -85,B 0,C 180,E1 -11967.89,E2 -11967.89} C_VEL
LIN {X 0,Y 381.877,Z 470.997,A -85,B 0,C 180,E1 -11968.945,E2 -11968.945} C_VEL
LIN {X 0,Y 381.909,Z 471.283,A -85,B 0,C 180,E1 -11970,E2 -11970} C_VEL
LIN {X 0,Y 381.85,Z 471.156,A -85,B 0,C 180,E1 -11971.054,E2 -11971.054} C_VEL
LIN {X 0,Y 381.859,Z 470.607,A -85,B 0,C 180,E1 -11972.109,E2 -11972.109} C_VEL
LIN {X 0,Y 381.798,Z 469.609,A -85,B 0,C 180,E1 -11973.165,E2 -11973.165} C_VEL
LIN {X 0,Y 381.723,Z 468.198,A -85,B 0,C 180,E1 -11974.223,E2 -11974.223} C_VEL
LIN {X 0,Y 381.708,Z 464.528,A -85,B 0,C 180,E1 -11976.147,E2 -11976.147} C_VEL
LIN {X 0,Y 381.879,Z 459.681,A -85,B 0,C 180,E1 -11977.933,E2 -11977.933} C_VEL
LIN {X 0,Y 382.197,Z 453.054,A -85,B 0,C 180,E1 -11979.793,E2 -11979.793} C_VEL
LIN {X 0,Y 382.765,Z 445.895,A -85,B 0,C 180,E1 -11981.384,E2 -11981.384} C_VEL
LIN {X 0,Y 383.531,Z 436.966,A -85,B 0,C 180,E1 -11982.972,E2 -11982.972} C_VEL
LIN {X 0,Y 384.382,Z 427.418,A -85,B 0,C 180,E1 -11984.35,E2 -11984.35} C_VEL
LIN {X 0,Y 385.449,Z 416.68,A -85,B 0,C 180,E1 -11985.601,E2 -11985.601} C_VEL
LIN {X 0,Y 386.518,Z 405.428,A -85,B 0,C 180,E1 -11986.641,E2 -11986.641} C_VEL
LIN {X 0,Y 387.59,Z 392.913,A -85,B 0,C 180,E1 -11987.545,E2 -11987.545} C_VEL
LIN {X 0,Y 388.582,Z 380.336,A -85,B 0,C 180,E1 -11988.213,E2 -11988.213} C_VEL
LIN {X 0,Y 389.297,Z 367.373,A -85,B 0,C 180,E1 -11988.689,E2 -11988.689} C_VEL
LIN {X 0,Y 389.851,Z 340.141,A -85,B 0,C 180,E1 -11989.288,E2 -11989.288} C_VEL
LIN {X 0,Y 390.691,Z 292.444,A -85,B 0,C 180,E1 -11990.287,E2 -11990.287} C_VEL
LIN {X 0,Y 387.844,Z 270.169,A -85,B 0,C 180,E1 -11990.973,E2 -11990.973} C_VEL
LIN {X 0,Y 385.251,Z 254.832,A -85,B 0,C 180,E1 -11991.506,E2 -11991.506} C_VEL
LIN {X 0,Y 386.687,Z 235.97,A -85,B 0,C 180,E1 -11994.996,E2 -11994.996} C_VEL
LIN {X 0,Y 387.349,Z 226.982,A -85,B 0,C 180,E1 -11996.683,E2 -11996.683} C_VEL
LIN {X 0,Y 385.6,Z 217.482,A -85,B 0,C 180,E1 -11998.671,E2 -11998.671} C_VEL
LIN {X 0,Y 382.995,Z 206.783,A -85,B 0,C 180,E1 -12001.071,E2 -12001.071} C_VEL
LIN {X 0,Y 383.018,Z 206.777,A -85,B 0,C 180,E1 -12004.668,E2 -12004.668} C_VEL
LIN {X 0,Y 382.994,Z 206.776,A -85,B 0,C 180,E1 -12007.902,E2 -12007.902} C_VEL
LIN {X 0,Y 382.963,Z 206.78,A -85,B 0,C 180,E1 -12011.35,E2 -12011.35} C_VEL
LIN {X 0,Y 382.995,Z 206.778,A -85,B 0,C 180,E1 -12014.303,E2 -12014.303} C_VEL
LIN {X 0,Y 383.01,Z 206.77,A -85,B 0,C 180,E1 -12017.24,E2 -12017.24} C_VEL
LIN {X 0,Y 382.986,Z 206.778,A -85,B 0,C 180,E1 -12020.418,E2 -12020.418} C_VEL
LIN {X 0,Y 383.024,Z 206.776,A -85,B 0,C 180,E1 -12024.044,E2 -12024.044} C_VEL
LIN {X 0,Y 382.987,Z 206.775,A -85,B 0,C 180,E1 -12027.578,E2 -12027.578} C_VEL
LIN {X 0,Y 382.98,Z 206.777,A -85,B 0,C 180,E1 -12030.299,E2 -12030.299} C_VEL
LIN {X 0,Y 383.022,Z 206.772,A -85,B 0,C 180,E1 -12034.038,E2 -12034.038} C_VEL
LIN {X 0,Y 382.991,Z 206.775,A -85,B 0,C 180,E1 -12037.334,E2 -12037.334} C_VEL
LIN {X 0,Y 383.058,Z 206.768,A -85,B 0,C 180,E1 -12040.716,E2 -12040.716} C_VEL
LIN {X 0,Y 383.08,Z 206.767,A -85,B 0,C 180,E1 -12044.027,E2 -12044.027} C_VEL
LIN {X 0,Y 383.136,Z 206.76,A -85,B 0,C 180,E1 -12047.284,E2 -12047.284} C_VEL
LIN {X 0,Y 383.151,Z 206.754,A -85,B 0,C 180,E1 -12050.498,E2 -12050.498} C_VEL
LIN {X 0,Y 383.28,Z 206.74,A -85,B 0,C 180,E1 -12053.684,E2 -12053.684} C_VEL
LIN {X 0,Y 383.385,Z 206.728,A -85,B 0,C 180,E1 -12057.899,E2 -12057.899} C_VEL
LIN {X 0,Y 383.518,Z 206.712,A -85,B 0,C 180,E1 -12060,E2 -12060} C_VEL
LIN {X 0,Y 383.246,Z 206.747,A -85,B 0,C 180,E1 -12063.154,E2 -12063.154} C_VEL
LIN {X 0,Y 383.242,Z 206.745,A -85,B 0,C 180,E1 -12066.472,E2 -12066.472} C_VEL
LIN {X 0,Y 383.143,Z 206.762,A -85,B 0,C 180,E1 -12069.502,E2 -12069.502} C_VEL
LIN {X 0,Y 383.125,Z 206.768,A -85,B 0,C 180,E1 -12073.536,E2 -12073.536} C_VEL
LIN {X 0,Y 383.1,Z 206.766,A -85,B 0,C 180,E1 -12076.383,E2 -12076.383} C_VEL
LIN {X 0,Y 384.205,Z 209.764,A -85,B 0,C 180,E1 -12076.556,E2 -12076.556} C_VEL
LIN {X 0,Y 390.625,Z 224.185,A -85,B 0,C 180,E1 -12077.344,E2 -12077.344} C_VEL
LIN {X 0,Y 391.955,Z 227.68,A -85,B 0,C 180,E1 -12077.513,E2 -12077.513} C_VEL
LIN {X 0,Y 390.112,Z 313.497,A -85,B 0,C 180,E1 -12079.331,E2 -12079.331} C_VEL
LIN {X 0,Y 389.712,Z 326.31,A -85,B 0,C 180,E1 -12079.798,E2 -12079.798} C_VEL
LIN {X 0,Y 389.113,Z 339.106,A -85,B 0,C 180,E1 -12080.477,E2 -12080.477} C_VEL
LIN {X 0,Y 388.28,Z 351.428,A -85,B 0,C 180,E1 -12081.363,E2 -12081.363} C_VEL
LIN {X 0,Y 387.438,Z 362.487,A -85,B 0,C 180,E1 -12082.391,E2 -12082.391} C_VEL
LIN {X 0,Y 386.528,Z 372.734,A -85,B 0,C 180,E1 -12083.579,E2 -12083.579} C_VEL
LIN {X 0,Y 385.682,Z 381.164,A -85,B 0,C 180,E1 -12084.779,E2 -12084.779} C_VEL
LIN {X 0,Y 384.823,Z 389.44,A -85,B 0,C 180,E1 -12086.223,E2 -12086.223} C_VEL
LIN {X 0,Y 383.992,Z 396.833,A -85,B 0,C 180,E1 -12087.821,E2 -12087.821} C_VEL
LIN {X 0,Y 383.411,Z 402.519,A -85,B 0,C 180,E1 -12089.362,E2 -12089.362} C_VEL
LIN {X 0,Y 382.865,Z 407.093,A -85,B 0,C 180,E1 -12090.929,E2 -12090.929} C_VEL
LIN {X 0,Y 382.393,Z 411.218,A -85,B 0,C 180,E1 -12092.845,E2 -12092.845} C_VEL
LIN {X 0,Y 382.068,Z 413.854,A -85,B 0,C 180,E1 -12094.766,E2 -12094.766} C_VEL
LIN {X 0,Y 381.899,Z 414.899,A -85,B 0,C 180,E1 -12096.078,E2 -12096.078} C_VEL
LIN {X 0,Y 381.796,Z 415.291,A -85,B 0,C 180,E1 -12097.671,E2 -12097.671} C_VEL
LIN {X 0,Y 381.812,Z 414.693,A -85,B 0,C 180,E1 -12099.368,E2 -12099.368} C_VEL
LIN {X 0,Y 381.948,Z 412.443,A -85,B 0,C 180,E1 -12101.484,E2 -12101.484} C_VEL
LIN {X 0,Y 382.178,Z 410.057,A -85,B 0,C 180,E1 -12102.875,E2 -12102.875} C_VEL
LIN {X 0,Y 382.423,Z 406.82,A -85,B 0,C 180,E1 -12104.295,E2 -12104.295} C_VEL
LIN {X 0,Y 382.817,Z 401.35,A -85,B 0,C 180,E1 -12106.101,E2 -12106.101} C_VEL
LIN {X 0,Y 383.266,Z 395.717,A -85,B 0,C 180,E1 -12107.567,E2 -12107.567} C_VEL
LIN {X 0,Y 383.947,Z 387.565,A -85,B 0,C 180,E1 -12109.266,E2 -12109.266} C_VEL
LIN {X 0,Y 384.691,Z 378.552,A -85,B 0,C 180,E1 -12110.76,E2 -12110.76} C_VEL
LIN {X 0,Y 385.426,Z 369.146,A -85,B 0,C 180,E1 -12112.025,E2 -12112.025} C_VEL
LIN {X 0,Y 386.149,Z 358.326,A -85,B 0,C 180,E1 -12113.208,E2 -12113.208} C_VEL
LIN {X 0,Y 386.934,Z 346.465,A -85,B 0,C 180,E1 -12114.223,E2 -12114.223} C_VEL
LIN {X 0,Y 387.52,Z 334.728,A -85,B 0,C 180,E1 -12115.002,E2 -12115.002} C_VEL
LIN {X 0,Y 387.937,Z 321.846,A -85,B 0,C 180,E1 -12115.637,E2 -12115.637} C_VEL
LIN {X 0,Y 388.255,Z 308.407,A -85,B 0,C 180,E1 -12116.061,E2 -12116.061} C_VEL
LIN {X 0,Y 389.705,Z 225.097,A -85,B 0,C 180,E1 -12117.747,E2 -12117.747} C_VEL
LIN {X 0,Y 383.014,Z 206.776,A -85,B 0,C 180,E1 -12118.47,E2 -12118.47} C_VEL
LIN {X 0,Y 383.03,Z 206.771,A -85,B 0,C 180,E1 -12121.73,E2 -12121.73} C_VEL
LIN {X 0,Y 383.049,Z 206.773,A -85,B 0,C 180,E1 -12125.04,E2 -12125.04} C_VEL
LIN {X 0,Y 382.992,Z 206.776,A -85,B 0,C 180,E1 -12128.469,E2 -12128.469} C_VEL
LIN {X 0,Y 383.053,Z 206.767,A -85,B 0,C 180,E1 -12131.826,E2 -12131.826} C_VEL
LIN {X 0,Y 383.111,Z 206.763,A -85,B 0,C 180,E1 -12135.119,E2 -12135.119} C_VEL
LIN {X 0,Y 383.098,Z 206.763,A -85,B 0,C 180,E1 -12138.358,E2 -12138.358} C_VEL
LIN {X 0,Y 383.221,Z 206.746,A -85,B 0,C 180,E1 -12142.022,E2 -12142.022} C_VEL
LIN {X 0,Y 383.189,Z 206.755,A -85,B 0,C 180,E1 -12144.739,E2 -12144.739} C_VEL
LIN {X 0,Y 383.385,Z 206.726,A -85,B 0,C 180,E1 -12147.899,E2 -12147.899} C_VEL
LIN {X 0,Y 383.443,Z 206.718,A -85,B 0,C 180,E1 -12150.3,E2 -12150.3} C_VEL
LIN {X 0,Y 382.603,Z 206.824,A -85,B 0,C 180,E1 -12151.176,E2 -12151.176} C_VEL
LIN {X 0,Y 379.552,Z 207.208,A -85,B 0,C 180,E1 -12152.596,E2 -12152.596} C_VEL
LIN {X 0,Y 377.102,Z 207.512,A -85,B 0,C 180,E1 -12153.745,E2 -12153.745} C_VEL
LIN {X 0,Y 376.128,Z 207.633,A -85,B 0,C 180,E1 -12154.636,E2 -12154.636} C_VEL
LIN {X 0,Y 376.085,Z 207.635,A -85,B 0,C 180,E1 -12154.937,E2 -12154.937} C_VEL
LIN {X 0,Y 376.17,Z 207.624,A -85,B 0,C 180,E1 -12157.515,E2 -12157.515} C_VEL
LIN {X 0,Y 376.084,Z 207.636,A -85,B 0,C 180,E1 -12160.771,E2 -12160.771} C_VEL
LIN {X 0,Y 376.067,Z 207.642,A -85,B 0,C 180,E1 -12164.061,E2 -12164.061} C_VEL
LIN {X 0,Y 376.046,Z 207.641,A -85,B 0,C 180,E1 -12167.608,E2 -12167.608} C_VEL
LIN {X 0,Y 375.98,Z 207.648,A -85,B 0,C 180,E1 -12170.832,E2 -12170.832} C_VEL
LIN {X 0,Y 375.979,Z 207.651,A -85,B 0,C 180,E1 -12174.283,E2 -12174.283} C_VEL
LIN {X 0,Y 375.937,Z 207.659,A -85,B 0,C 180,E1 -12177.864,E2 -12177.864} C_VEL
LIN {X 0,Y 375.959,Z 207.655,A -85,B 0,C 180,E1 -12181.562,E2 -12181.562} C_VEL
LIN {X 0,Y 375.959,Z 207.654,A -85,B 0,C 180,E1 -12185.416,E2 -12185.416} C_VEL
LIN {X 0,Y 375.938,Z 207.654,A -85,B 0,C 180,E1 -12188.263,E2 -12188.263} C_VEL
LIN {X 0,Y 375.924,Z 207.66,A -85,B 0,C 180,E1 -12191.599,E2 -12191.599} C_VEL
LIN {X 0,Y 375.928,Z 207.659,A -85,B 0,C 180,E1 -12195.269,E2 -12195.269} C_VEL
LIN {X 0,Y 375.92,Z 207.655,A -85,B 0,C 180,E1 -12198.402,E2 -12198.402} C_VEL
LIN {X 0,Y 375.956,Z 207.652,A -85,B 0,C 180,E1 -12201.91,E2 -12201.91} C_VEL
LIN {X 0,Y 375.982,Z 207.652,A -85,B 0,C 180,E1 -12205.333,E2 -12205.333} C_VEL
LIN {X 0,Y 375.96,Z 207.651,A -85,B 0,C 180,E1 -12208.438,E2 -12208.438} C_VEL
LIN {X 0,Y 375.931,Z 207.654,A -85,B 0,C 180,E1 -12212.136,E2 -12212.136} C_VEL
LIN {X 0,Y 375.975,Z 207.649,A -85,B 0,C 180,E1 -12215.717,E2 -12215.717} C_VEL
LIN {X 0,Y 376.001,Z 207.648,A -85,B 0,C 180,E1 -12219.198,E2 -12219.198} C_VEL
LIN {X 0,Y 376.035,Z 207.645,A -85,B 0,C 180,E1 -12222.6,E2 -12222.6} C_VEL
LIN {X 0,Y 376.093,Z 207.637,A -85,B 0,C 180,E1 -12226.343,E2 -12226.343} C_VEL
LIN {X 0,Y 376.116,Z 207.634,A -85,B 0,C 180,E1 -12230.319,E2 -12230.319} C_VEL
LIN {X 0,Y 376.203,Z 207.62,A -85,B 0,C 180,E1 -12233.564,E2 -12233.564} C_VEL
LIN {X 0,Y 376.348,Z 207.603,A -85,B 0,C 180,E1 -12237.86,E2 -12237.86} C_VEL
LIN {X 0,Y 376.266,Z 207.612,A -85,B 0,C 180,E1 -12241.07,E2 -12241.07} C_VEL
LIN {X 0,Y 376.341,Z 207.607,A -85,B 0,C 180,E1 -12242.141,E2 -12242.141} C_VEL
LIN {X 0,Y 376.201,Z 207.624,A -85,B 0,C 180,E1 -12246.436,E2 -12246.436} C_VEL
LIN {X 0,Y 376.116,Z 207.633,A -85,B 0,C 180,E1 -12249.682,E2 -12249.682} C_VEL
LIN {X 0,Y 376.093,Z 207.636,A -85,B 0,C 180,E1 -12253.658,E2 -12253.658} C_VEL
LIN {X 0,Y 376.015,Z 207.646,A -85,B 0,C 180,E1 -12257.592,E2 -12257.592} C_VEL
LIN {X 0,Y 375.982,Z 207.647,A -85,B 0,C 180,E1 -12260.832,E2 -12260.832} C_VEL
LIN {X 0,Y 375.938,Z 207.655,A -85,B 0,C 180,E1 -12264.285,E2 -12264.285} C_VEL
LIN {X 0,Y 375.922,Z 207.655,A -85,B 0,C 180,E1 -12266.66,E2 -12266.66} C_VEL
LIN {X 0,Y 375.919,Z 207.656,A -85,B 0,C 180,E1 -12269.084,E2 -12269.084} C_VEL
LIN {X 0,Y 375.959,Z 207.656,A -85,B 0,C 180,E1 -12271.562,E2 -12271.562} C_VEL
LIN {X 0,Y 375.958,Z 207.656,A -85,B 0,C 180,E1 -12275.416,E2 -12275.416} C_VEL
LIN {X 0,Y 375.938,Z 207.653,A -85,B 0,C 180,E1 -12278.263,E2 -12278.263} C_VEL
LIN {X 0,Y 375.917,Z 207.66,A -85,B 0,C 180,E1 -12281.597,E2 -12281.597} C_VEL
LIN {X 0,Y 375.923,Z 207.656,A -85,B 0,C 180,E1 -12284.73,E2 -12284.73} C_VEL
LIN {X 0,Y 375.927,Z 207.656,A -85,B 0,C 180,E1 -12287.699,E2 -12287.699} C_VEL
LIN {X 0,Y 375.938,Z 207.654,A -85,B 0,C 180,E1 -12290.534,E2 -12290.534} C_VEL
LIN {X 0,Y 375.961,Z 207.652,A -85,B 0,C 180,E1 -12293.497,E2 -12293.497} C_VEL
LIN {X 0,Y 375.959,Z 207.652,A -85,B 0,C 180,E1 -12295.888,E2 -12295.888} C_VEL
LIN {X 0,Y 375.962,Z 207.655,A -85,B 0,C 180,E1 -12299.034,E2 -12299.034} C_VEL
LIN {X 0,Y 378.625,Z 220.053,A -85,B 0,C 180,E1 -12301.749,E2 -12301.749} C_VEL
LIN {X 0,Y 380.01,Z 227.844,A -85,B 0,C 180,E1 -12303.394,E2 -12303.394} C_VEL
LIN {X 0,Y 378.63,Z 245.186,A -85,B 0,C 180,E1 -12306.769,E2 -12306.769} C_VEL
LIN {X 0,Y 377.732,Z 257.84,A -85,B 0,C 180,E1 -12309.213,E2 -12309.213} C_VEL
LIN {X 0,Y 382.207,Z 294.74,A -85,B 0,C 180,E1 -12310.225,E2 -12310.225} C_VEL
LIN {X 0,Y 380.928,Z 367.732,A -85,B 0,C 180,E1 -12311.755,E2 -12311.755} C_VEL
LIN {X 0,Y 380.262,Z 381.887,A -85,B 0,C 180,E1 -12312.279,E2 -12312.279} C_VEL
LIN {X 0,Y 379.45,Z 394.461,A -85,B 0,C 180,E1 -12312.97,E2 -12312.97} C_VEL
LIN {X 0,Y 378.593,Z 406.139,A -85,B 0,C 180,E1 -12313.832,E2 -12313.832} C_VEL
LIN {X 0,Y 377.589,Z 417.463,A -85,B 0,C 180,E1 -12314.895,E2 -12314.895} C_VEL
LIN {X 0,Y 376.8,Z 427.459,A -85,B 0,C 180,E1 -12316.071,E2 -12316.071} C_VEL
LIN {X 0,Y 376.114,Z 436.11,A -85,B 0,C 180,E1 -12317.317,E2 -12317.317} C_VEL
LIN {X 0,Y 375.58,Z 443.88,A -85,B 0,C 180,E1 -12318.668,E2 -12318.668} C_VEL
LIN {X 0,Y 375.071,Z 451.48,A -85,B 0,C 180,E1 -12320.291,E2 -12320.291} C_VEL
LIN {X 0,Y 374.822,Z 457.575,A -85,B 0,C 180,E1 -12321.916,E2 -12321.916} C_VEL
LIN {X 0,Y 374.71,Z 462.927,A -85,B 0,C 180,E1 -12323.754,E2 -12323.754} C_VEL
LIN {X 0,Y 374.664,Z 466.953,A -85,B 0,C 180,E1 -12325.697,E2 -12325.697} C_VEL
LIN {X 0,Y 374.735,Z 468.563,A -85,B 0,C 180,E1 -12326.774,E2 -12326.774} C_VEL
LIN {X 0,Y 374.807,Z 469.744,A -85,B 0,C 180,E1 -12327.85,E2 -12327.85} C_VEL
LIN {X 0,Y 374.801,Z 470.451,A -85,B 0,C 180,E1 -12328.925,E2 -12328.925} C_VEL
LIN {X 0,Y 374.828,Z 470.748,A -85,B 0,C 180,E1 -12330,E2 -12330} C_VEL
LIN {X 0,Y 374.775,Z 470.633,A -85,B 0,C 180,E1 -12331.074,E2 -12331.074} C_VEL
LIN {X 0,Y 374.789,Z 470.107,A -85,B 0,C 180,E1 -12332.149,E2 -12332.149} C_VEL
LIN {X 0,Y 374.7,Z 469.118,A -85,B 0,C 180,E1 -12333.225,E2 -12333.225} C_VEL
LIN {X 0,Y 374.644,Z 467.717,A -85,B 0,C 180,E1 -12334.303,E2 -12334.303} C_VEL
LIN {X 0,Y 374.612,Z 464.409,A -85,B 0,C 180,E1 -12336.107,E2 -12336.107} C_VEL
LIN {X 0,Y 374.751,Z 460.834,A -85,B 0,C 180,E1 -12337.543,E2 -12337.543} C_VEL
LIN {X 0,Y 374.949,Z 455.718,A -85,B 0,C 180,E1 -12339.167,E2 -12339.167} C_VEL
LIN {X 0,Y 375.373,Z 449.312,A -85,B 0,C 180,E1 -12340.791,E2 -12340.791} C_VEL
LIN {X 0,Y 376.19,Z 441.386,A -85,B 0,C 180,E1 -12342.406,E2 -12342.406} C_VEL
LIN {X 0,Y 376.917,Z 433.297,A -85,B 0,C 180,E1 -12343.753,E2 -12343.753} C_VEL
LIN {X 0,Y 377.869,Z 423.473,A -85,B 0,C 180,E1 -12345.093,E2 -12345.093} C_VEL
LIN {X 0,Y 378.983,Z 412.63,A -85,B 0,C 180,E1 -12346.289,E2 -12346.289} C_VEL
LIN {X 0,Y 380.034,Z 402.211,A -85,B 0,C 180,E1 -12347.211,E2 -12347.211} C_VEL
LIN {X 0,Y 381.113,Z 389.909,A -85,B 0,C 180,E1 -12348.061,E2 -12348.061} C_VEL
LIN {X 0,Y 382.129,Z 376.457,A -85,B 0,C 180,E1 -12348.74,E2 -12348.74} C_VEL
LIN {X 0,Y 382.832,Z 364.212,A -85,B 0,C 180,E1 -12349.156,E2 -12349.156} C_VEL
LIN {X 0,Y 384.208,Z 293.424,A -85,B 0,C 180,E1 -12350.679,E2 -12350.679} C_VEL
LIN {X 0,Y 381.392,Z 271.487,A -85,B 0,C 180,E1 -12351.374,E2 -12351.374} C_VEL
LIN {X 0,Y 378.457,Z 254.151,A -85,B 0,C 180,E1 -12352.005,E2 -12352.005} C_VEL
LIN {X 0,Y 379.896,Z 235.786,A -85,B 0,C 180,E1 -12355.475,E2 -12355.475} C_VEL
LIN {X 0,Y 380.506,Z 228.413,A -85,B 0,C 180,E1 -12356.883,E2 -12356.883} C_VEL
LIN {X 0,Y 378.436,Z 217.659,A -85,B 0,C 180,E1 -12359.209,E2 -12359.209} C_VEL
LIN {X 0,Y 375.961,Z 207.656,A -85,B 0,C 180,E1 -12361.506,E2 -12361.506} C_VEL
LIN {X 0,Y 375.957,Z 207.653,A -85,B 0,C 180,E1 -12365.415,E2 -12365.415} C_VEL
LIN {X 0,Y 375.936,Z 207.657,A -85,B 0,C 180,E1 -12368.263,E2 -12368.263} C_VEL
LIN {X 0,Y 375.919,Z 207.657,A -85,B 0,C 180,E1 -12371.598,E2 -12371.598} C_VEL
LIN {X 0,Y 375.926,Z 207.656,A -85,B 0,C 180,E1 -12374.731,E2 -12374.731} C_VEL
LIN {X 0,Y 375.926,Z 207.653,A -85,B 0,C 180,E1 -12377.699,E2 -12377.699} C_VEL
LIN {X 0,Y 375.935,Z 207.657,A -85,B 0,C 180,E1 -12380.534,E2 -12380.534} C_VEL
LIN {X 0,Y 375.963,Z 207.652,A -85,B 0,C 180,E1 -12383.496,E2 -12383.496} C_VEL
LIN {X 0,Y 375.96,Z 207.652,A -85,B 0,C 180,E1 -12385.888,E2 -12385.888} C_VEL
LIN {X 0,Y 375.962,Z 207.653,A -85,B 0,C 180,E1 -12389.687,E2 -12389.687} C_VEL
LIN {X 0,Y 375.94,Z 207.652,A -85,B 0,C 180,E1 -12393.342,E2 -12393.342} C_VEL
LIN {X 0,Y 375.977,Z 207.648,A -85,B 0,C 180,E1 -12396.887,E2 -12396.887} C_VEL
LIN {X 0,Y 375.997,Z 207.65,A -85,B 0,C 180,E1 -12400.339,E2 -12400.339} C_VEL
LIN {X 0,Y 376.025,Z 207.646,A -85,B 0,C 180,E1 -12403.719,E2 -12403.719} C_VEL
LIN {X 0,Y 376.103,Z 207.634,A -85,B 0,C 180,E1 -12407.042,E2 -12407.042} C_VEL
LIN {X 0,Y 376.119,Z 207.631,A -85,B 0,C 180,E1 -12410.318,E2 -12410.318} C_VEL
LIN {X 0,Y 376.238,Z 207.618,A -85,B 0,C 180,E1 -12413.565,E2 -12413.565} C_VEL
LIN {X 0,Y 376.351,Z 207.604,A -85,B 0,C 180,E1 -12417.86,E2 -12417.86} C_VEL
LIN {X 0,Y 376.487,Z 207.588,A -85,B 0,C 180,E1 -12420,E2 -12420} C_VEL
LIN {X 0,Y 376.184,Z 207.627,A -85,B 0,C 180,E1 -12423.213,E2 -12423.213} C_VEL
LIN {X 0,Y 376.212,Z 207.621,A -85,B 0,C 180,E1 -12426.456,E2 -12426.456} C_VEL
LIN {X 0,Y 376.113,Z 207.638,A -85,B 0,C 180,E1 -12429.682,E2 -12429.682} C_VEL
LIN {X 0,Y 376.088,Z 207.644,A -85,B 0,C 180,E1 -12433.657,E2 -12433.657} C_VEL
LIN {X 0,Y 376.086,Z 207.828,A -85,B 0,C 180,E1 -12435.896,E2 -12435.896} C_VEL
LIN {X 0,Y 377.223,Z 210.738,A -85,B 0,C 180,E1 -12436.055,E2 -12436.055} C_VEL
LIN {X 0,Y 383.865,Z 225.295,A -85,B 0,C 180,E1 -12436.902,E2 -12436.902} C_VEL
LIN {X 0,Y 385.55,Z 229.906,A -85,B 0,C 180,E1 -12437.128,E2 -12437.128} C_VEL
LIN {X 0,Y 383.556,Z 314.203,A -85,B 0,C 180,E1 -12438.945,E2 -12438.945} C_VEL
LIN {X 0,Y 383.137,Z 326.886,A -85,B 0,C 180,E1 -12439.416,E2 -12439.416} C_VEL
LIN {X 0,Y 382.484,Z 340.121,A -85,B 0,C 180,E1 -12440.133,E2 -12440.133} C_VEL
LIN {X 0,Y 381.605,Z 352.436,A -85,B 0,C 180,E1 -12441.047,E2 -12441.047} C_VEL
LIN {X 0,Y 380.645,Z 363.872,A -85,B 0,C 180,E1 -12442.142,E2 -12442.142} C_VEL
LIN {X 0,Y 379.728,Z 373.578,A -85,B 0,C 180,E1 -12443.304,E2 -12443.304} C_VEL
LIN {X 0,Y 378.782,Z 382.458,A -85,B 0,C 180,E1 -12444.611,E2 -12444.611} C_VEL
LIN {X 0,Y 377.793,Z 391.3,A -85,B 0,C 180,E1 -12446.22,E2 -12446.22} C_VEL
LIN {X 0,Y 376.994,Z 398.182,A -85,B 0,C 180,E1 -12447.778,E2 -12447.778} C_VEL
LIN {X 0,Y 376.383,Z 403.724,A -85,B 0,C 180,E1 -12449.351,E2 -12449.351} C_VEL
LIN {X 0,Y 375.769,Z 408.483,A -85,B 0,C 180,E1 -12451.088,E2 -12451.088} C_VEL
LIN {X 0,Y 375.312,Z 412.078,A -85,B 0,C 180,E1 -12452.891,E2 -12452.891} C_VEL
LIN {X 0,Y 375.037,Z 414.206,A -85,B 0,C 180,E1 -12454.459,E2 -12454.459} C_VEL
LIN {X 0,Y 374.797,Z 415.547,A -85,B 0,C 180,E1 -12456.263,E2 -12456.263} C_VEL
LIN {X 0,Y 374.706,Z 415.708,A -85,B 0,C 180,E1 -12458.239,E2 -12458.239} C_VEL
LIN {X 0,Y 374.724,Z 414.912,A -85,B 0,C 180,E1 -12459.74,E2 -12459.74} C_VEL
LIN {X 0,Y 374.876,Z 413.077,A -85,B 0,C 180,E1 -12461.418,E2 -12461.418} C_VEL
LIN {X 0,Y 375.133,Z 410.278,A -85,B 0,C 180,E1 -12463.059,E2 -12463.059} C_VEL
LIN {X 0,Y 375.437,Z 406.532,A -85,B 0,C 180,E1 -12464.656,E2 -12464.656} C_VEL
LIN {X 0,Y 375.852,Z 400.932,A -85,B 0,C 180,E1 -12466.469,E2 -12466.469} C_VEL
LIN {X 0,Y 376.355,Z 394.626,A -85,B 0,C 180,E1 -12468.068,E2 -12468.068} C_VEL
LIN {X 0,Y 377.017,Z 387.214,A -85,B 0,C 180,E1 -12469.58,E2 -12469.58} C_VEL
LIN {X 0,Y 377.776,Z 378.038,A -85,B 0,C 180,E1 -12471.092,E2 -12471.092} C_VEL
LIN {X 0,Y 378.588,Z 368.191,A -85,B 0,C 180,E1 -12472.407,E2 -12472.407} C_VEL
LIN {X 0,Y 379.255,Z 358.51,A -85,B 0,C 180,E1 -12473.462,E2 -12473.462} C_VEL
LIN {X 0,Y 380.038,Z 347.04,A -85,B 0,C 180,E1 -12474.458,E2 -12474.458} C_VEL
LIN {X 0,Y 380.737,Z 333.686,A -85,B 0,C 180,E1 -12475.347,E2 -12475.347} C_VEL
LIN {X 0,Y 381.167,Z 320.696,A -85,B 0,C 180,E1 -12475.964,E2 -12475.964} C_VEL
LIN {X 0,Y 381.465,Z 306.846,A -85,B 0,C 180,E1 -12476.384,E2 -12476.384} C_VEL
LIN {X 0,Y 383,Z 227.179,A -85,B 0,C 180,E1 -12478.02,E2 -12478.02} C_VEL
LIN {X 0,Y 377.529,Z 212.182,A -85,B 0,C 180,E1 -12478.615,E2 -12478.615} C_VEL
LIN {X 0,Y 375.972,Z 207.653,A -85,B 0,C 180,E1 -12478.804,E2 -12478.804} C_VEL
LIN {X 0,Y 375.983,Z 207.647,A -85,B 0,C 180,E1 -12482.141,E2 -12482.141} C_VEL
LIN {X 0,Y 376.004,Z 207.646,A -85,B 0,C 180,E1 -12484.539,E2 -12484.539} C_VEL
LIN {X 0,Y 375.957,Z 207.651,A -85,B 0,C 180,E1 -12488.046,E2 -12488.046} C_VEL
LIN {X 0,Y 376.003,Z 207.646,A -85,B 0,C 180,E1 -12491.473,E2 -12491.473} C_VEL
LIN {X 0,Y 376.059,Z 207.644,A -85,B 0,C 180,E1 -12494.833,E2 -12494.833} C_VEL
LIN {X 0,Y 376.05,Z 207.64,A -85,B 0,C 180,E1 -12498.137,E2 -12498.137} C_VEL
LIN {X 0,Y 376.174,Z 207.624,A -85,B 0,C 180,E1 -12501.969,E2 -12501.969} C_VEL
LIN {X 0,Y 376.16,Z 207.632,A -85,B 0,C 180,E1 -12504.64,E2 -12504.64} C_VEL
LIN {X 0,Y 376.351,Z 207.602,A -85,B 0,C 180,E1 -12507.86,E2 -12507.86} C_VEL
LIN {X 0,Y 376.421,Z 207.593,A -85,B 0,C 180,E1 -12510.263,E2 -12510.263} C_VEL
LIN {X 0,Y 376.345,Z 207.605,A -85,B 0,C 180,E1 -12512.141,E2 -12512.141} C_VEL
LIN {X 0,Y 376.085,Z 207.635,A -85,B 0,C 180,E1 -12514.937,E2 -12514.937} C_VEL
LIN {X 0,Y 375.509,Z 207.709,A -85,B 0,C 180,E1 -12515.832,E2 -12515.832} C_VEL
LIN {X 0,Y 372.659,Z 208.061,A -85,B 0,C 180,E1 -12517.287,E2 -12517.287} C_VEL
LIN {X 0,Y 370.193,Z 208.373,A -85,B 0,C 180,E1 -12518.464,E2 -12518.464} C_VEL
LIN {X 0,Y 369.139,Z 208.501,A -85,B 0,C 180,E1 -12519.375,E2 -12519.375} C_VEL
LIN {X 0,Y 369.06,Z 208.511,A -85,B 0,C 180,E1 -12519.683,E2 -12519.683} C_VEL
LIN {X 0,Y 369.039,Z 208.515,A -85,B 0,C 180,E1 -12523.773,E2 -12523.773} C_VEL
LIN {X 0,Y 369.003,Z 208.52,A -85,B 0,C 180,E1 -12527.769,E2 -12527.769} C_VEL
LIN {X 0,Y 368.911,Z 208.529,A -85,B 0,C 180,E1 -12531.221,E2 -12531.221} C_VEL
LIN {X 0,Y 368.936,Z 208.525,A -85,B 0,C 180,E1 -12534.777,E2 -12534.777} C_VEL
LIN {X 0,Y 368.918,Z 208.528,A -85,B 0,C 180,E1 -12538.442,E2 -12538.442} C_VEL
LIN {X 0,Y 368.912,Z 208.528,A -85,B 0,C 180,E1 -12540.988,E2 -12540.988} C_VEL
LIN {X 0,Y 368.938,Z 208.525,A -85,B 0,C 180,E1 -12544.854,E2 -12544.854} C_VEL
LIN {X 0,Y 368.879,Z 208.532,A -85,B 0,C 180,E1 -12548.634,E2 -12548.634} C_VEL
LIN {X 0,Y 368.875,Z 208.534,A -85,B 0,C 180,E1 -12552.008,E2 -12552.008} C_VEL
LIN {X 0,Y 368.881,Z 208.536,A -85,B 0,C 180,E1 -12555.176,E2 -12555.176} C_VEL
LIN {X 0,Y 368.872,Z 208.533,A -85,B 0,C 180,E1 -12558.176,E2 -12558.176} C_VEL
LIN {X 0,Y 368.879,Z 208.538,A -85,B 0,C 180,E1 -12561.366,E2 -12561.366} C_VEL
LIN {X 0,Y 368.939,Z 208.531,A -85,B 0,C 180,E1 -12565.147,E2 -12565.147} C_VEL
LIN {X 0,Y 368.932,Z 208.532,A -85,B 0,C 180,E1 -12569.047,E2 -12569.047} C_VEL
LIN {X 0,Y 368.87,Z 208.537,A -85,B 0,C 180,E1 -12572.789,E2 -12572.789} C_VEL
LIN {X 0,Y 368.952,Z 208.525,A -85,B 0,C 180,E1 -12576.421,E2 -12576.421} C_VEL
LIN {X 0,Y 368.938,Z 208.525,A -85,B 0,C 180,E1 -12579.947,E2 -12579.947} C_VEL
LIN {X 0,Y 368.971,Z 208.522,A -85,B 0,C 180,E1 -12583.399,E2 -12583.399} C_VEL
LIN {X 0,Y 369.061,Z 208.515,A -85,B 0,C 180,E1 -12586.79,E2 -12586.79} C_VEL
LIN {X 0,Y 369.066,Z 208.511,A -85,B 0,C 180,E1 -12590.132,E2 -12590.132} C_VEL
LIN {X 0,Y 369.164,Z 208.497,A -85,B 0,C 180,E1 -12593.441,E2 -12593.441} C_VEL
LIN {X 0,Y 369.311,Z 208.479,A -85,B 0,C 180,E1 -12597.819,E2 -12597.819} C_VEL
LIN {X 0,Y 369.235,Z 208.488,A -85,B 0,C 180,E1 -12601.091,E2 -12601.091} C_VEL
LIN {X 0,Y 369.305,Z 208.484,A -85,B 0,C 180,E1 -12602.181,E2 -12602.181} C_VEL
LIN {X 0,Y 369.162,Z 208.5,A -85,B 0,C 180,E1 -12606.559,E2 -12606.559} C_VEL
LIN {X 0,Y 369.066,Z 208.513,A -85,B 0,C 180,E1 -12609.868,E2 -12609.868} C_VEL
LIN {X 0,Y 369.041,Z 208.516,A -85,B 0,C 180,E1 -12613.772,E2 -12613.772} C_VEL
LIN {X 0,Y 368.98,Z 208.524,A -85,B 0,C 180,E1 -12617.756,E2 -12617.756} C_VEL
LIN {X 0,Y 368.912,Z 208.529,A -85,B 0,C 180,E1 -12621.221,E2 -12621.221} C_VEL
LIN {X 0,Y 368.913,Z 208.534,A -85,B 0,C 180,E1 -12623.875,E2 -12623.875} C_VEL
LIN {X 0,Y 368.867,Z 208.535,A -85,B 0,C 180,E1 -12627.211,E2 -12627.211} C_VEL
LIN {X 0,Y 368.897,Z 208.536,A -85,B 0,C 180,E1 -12629.692,E2 -12629.692} C_VEL
LIN {X 0,Y 368.899,Z 208.531,A -85,B 0,C 180,E1 -12633.043,E2 -12633.043} C_VEL
LIN {X 0,Y 368.918,Z 208.528,A -85,B 0,C 180,E1 -12636.197,E2 -12636.197} C_VEL
LIN {X 0,Y 368.876,Z 208.534,A -85,B 0,C 180,E1 -12638.957,E2 -12638.957} C_VEL
LIN {X 0,Y 368.866,Z 208.535,A -85,B 0,C 180,E1 -12642.006,E2 -12642.006} C_VEL
LIN {X 0,Y 368.876,Z 208.538,A -85,B 0,C 180,E1 -12645.175,E2 -12645.175} C_VEL
LIN {X 0,Y 368.871,Z 208.533,A -85,B 0,C 180,E1 -12648.175,E2 -12648.175} C_VEL
LIN {X 0,Y 368.88,Z 208.536,A -85,B 0,C 180,E1 -12651.366,E2 -12651.366} C_VEL
LIN {X 0,Y 368.933,Z 208.531,A -85,B 0,C 180,E1 -12655.146,E2 -12655.146} C_VEL
LIN {X 0,Y 368.962,Z 208.672,A -85,B 0,C 180,E1 -12658.785,E2 -12658.785} C_VEL
LIN {X 0,Y 371.834,Z 222.221,A -85,B 0,C 180,E1 -12661.801,E2 -12661.801} C_VEL
LIN {X 0,Y 373.044,Z 229.785,A -85,B 0,C 180,E1 -12663.42,E2 -12663.42} C_VEL
LIN {X 0,Y 371.524,Z 247.3,A -85,B 0,C 180,E1 -12666.888,E2 -12666.888} C_VEL
LIN {X 0,Y 370.786,Z 257.357,A -85,B 0,C 180,E1 -12668.866,E2 -12668.866} C_VEL
LIN {X 0,Y 375.364,Z 294.265,A -85,B 0,C 180,E1 -12669.909,E2 -12669.909} C_VEL
LIN {X 0,Y 374.076,Z 367.375,A -85,B 0,C 180,E1 -12671.48,E2 -12671.48} C_VEL
LIN {X 0,Y 373.369,Z 381.463,A -85,B 0,C 180,E1 -12672.012,E2 -12672.012} C_VEL
LIN {X 0,Y 372.54,Z 394.009,A -85,B 0,C 180,E1 -12672.715,E2 -12672.715} C_VEL
LIN {X 0,Y 371.603,Z 406.475,A -85,B 0,C 180,E1 -12673.66,E2 -12673.66} C_VEL
LIN {X 0,Y 370.573,Z 417.644,A -85,B 0,C 180,E1 -12674.743,E2 -12674.743} C_VEL
LIN {X 0,Y 369.762,Z 427.516,A -85,B 0,C 180,E1 -12675.945,E2 -12675.945} C_VEL
LIN {X 0,Y 368.992,Z 436.887,A -85,B 0,C 180,E1 -12677.347,E2 -12677.347} C_VEL
LIN {X 0,Y 368.445,Z 444.448,A -85,B 0,C 180,E1 -12678.725,E2 -12678.725} C_VEL
LIN {X 0,Y 367.963,Z 451.865,A -85,B 0,C 180,E1 -12680.379,E2 -12680.379} C_VEL
LIN {X 0,Y 367.758,Z 456.869,A -85,B 0,C 180,E1 -12681.759,E2 -12681.759} C_VEL
LIN {X 0,Y 367.64,Z 461.705,A -85,B 0,C 180,E1 -12683.413,E2 -12683.413} C_VEL
LIN {X 0,Y 367.642,Z 465.373,A -85,B 0,C 180,E1 -12685.065,E2 -12685.065} C_VEL
LIN {X 0,Y 367.642,Z 467.969,A -85,B 0,C 180,E1 -12686.712,E2 -12686.712} C_VEL
LIN {X 0,Y 367.737,Z 469.173,A -85,B 0,C 180,E1 -12687.809,E2 -12687.809} C_VEL
LIN {X 0,Y 367.727,Z 469.902,A -85,B 0,C 180,E1 -12688.905,E2 -12688.905} C_VEL
LIN {X 0,Y 367.75,Z 470.212,A -85,B 0,C 180,E1 -12690,E2 -12690} C_VEL
LIN {X 0,Y 367.703,Z 470.111,A -85,B 0,C 180,E1 -12691.095,E2 -12691.095} C_VEL
LIN {X 0,Y 367.72,Z 469.606,A -85,B 0,C 180,E1 -12692.19,E2 -12692.19} C_VEL
LIN {X 0,Y 367.603,Z 468.637,A -85,B 0,C 180,E1 -12693.288,E2 -12693.288} C_VEL
LIN {X 0,Y 367.566,Z 467.254,A -85,B 0,C 180,E1 -12694.386,E2 -12694.386} C_VEL
LIN {X 0,Y 367.516,Z 464.299,A -85,B 0,C 180,E1 -12696.067,E2 -12696.067} C_VEL
LIN {X 0,Y 367.678,Z 460.426,A -85,B 0,C 180,E1 -12697.689,E2 -12697.689} C_VEL
LIN {X 0,Y 367.9,Z 455.338,A -85,B 0,C 180,E1 -12699.345,E2 -12699.345} C_VEL
LIN {X 0,Y 368.366,Z 448.962,A -85,B 0,C 180,E1 -12700.999,E2 -12700.999} C_VEL
LIN {X 0,Y 369.226,Z 441.083,A -85,B 0,C 180,E1 -12702.644,E2 -12702.644} C_VEL
LIN {X 0,Y 369.993,Z 433.057,A -85,B 0,C 180,E1 -12704.015,E2 -12704.015} C_VEL
LIN {X 0,Y 370.991,Z 423.326,A -85,B 0,C 180,E1 -12705.379,E2 -12705.379} C_VEL
LIN {X 0,Y 372.178,Z 412.604,A -85,B 0,C 180,E1 -12706.595,E2 -12706.595} C_VEL
LIN {X 0,Y 373.422,Z 400.696,A -85,B 0,C 180,E1 -12707.667,E2 -12707.667} C_VEL
LIN {X 0,Y 374.566,Z 388.084,A -85,B 0,C 180,E1 -12708.53,E2 -12708.53} C_VEL
LIN {X 0,Y 375.597,Z 374.969,A -85,B 0,C 180,E1 -12709.185,E2 -12709.185} C_VEL
LIN {X 0,Y 376.263,Z 362.029,A -85,B 0,C 180,E1 -12709.61,E2 -12709.61} C_VEL
LIN {X 0,Y 377.692,Z 294.118,A -85,B 0,C 180,E1 -12711.097,E2 -12711.097} C_VEL
LIN {X 0,Y 375.178,Z 273.992,A -85,B 0,C 180,E1 -12711.754,E2 -12711.754} C_VEL
LIN {X 0,Y 372.131,Z 256.02,A -85,B 0,C 180,E1 -12712.417,E2 -12712.417} C_VEL
LIN {X 0,Y 371.71,Z 253.43,A -85,B 0,C 180,E1 -12712.538,E2 -12712.538} C_VEL
LIN {X 0,Y 373.213,Z 235.664,A -85,B 0,C 180,E1 -12715.965,E2 -12715.965} C_VEL
LIN {X 0,Y 373.683,Z 230.082,A -85,B 0,C 180,E1 -12717.057,E2 -12717.057} C_VEL
LIN {X 0,Y 371.778,Z 220.076,A -85,B 0,C 180,E1 -12719.26,E2 -12719.26} C_VEL
LIN {X 0,Y 368.91,Z 208.534,A -85,B 0,C 180,E1 -12722.008,E2 -12722.008} C_VEL
LIN {X 0,Y 368.929,Z 208.532,A -85,B 0,C 180,E1 -12725.001,E2 -12725.001} C_VEL
LIN {X 0,Y 368.877,Z 208.536,A -85,B 0,C 180,E1 -12728.634,E2 -12728.634} C_VEL
LIN {X 0,Y 368.871,Z 208.535,A -85,B 0,C 180,E1 -12732.007,E2 -12732.007} C_VEL
LIN {X 0,Y 368.879,Z 208.532,A -85,B 0,C 180,E1 -12735.175,E2 -12735.175} C_VEL
LIN {X 0,Y 368.87,Z 208.534,A -85,B 0,C 180,E1 -12738.176,E2 -12738.176} C_VEL
LIN {X 0,Y 368.877,Z 208.535,A -85,B 0,C 180,E1 -12741.366,E2 -12741.366} C_VEL
LIN {X 0,Y 368.936,Z 208.525,A -85,B 0,C 180,E1 -12745.146,E2 -12745.146} C_VEL
LIN {X 0,Y 368.929,Z 208.528,A -85,B 0,C 180,E1 -12749.046,E2 -12749.046} C_VEL
LIN {X 0,Y 368.878,Z 208.532,A -85,B 0,C 180,E1 -12752.79,E2 -12752.79} C_VEL
LIN {X 0,Y 368.928,Z 208.527,A -85,B 0,C 180,E1 -12756.119,E2 -12756.119} C_VEL
LIN {X 0,Y 368.936,Z 208.526,A -85,B 0,C 180,E1 -12759.947,E2 -12759.947} C_VEL
LIN {X 0,Y 368.968,Z 208.521,A -85,B 0,C 180,E1 -12763.398,E2 -12763.398} C_VEL
LIN {X 0,Y 369.058,Z 208.511,A -85,B 0,C 180,E1 -12766.79,E2 -12766.79} C_VEL
LIN {X 0,Y 369.067,Z 208.51,A -85,B 0,C 180,E1 -12770.132,E2 -12770.132} C_VEL
LIN {X 0,Y 369.199,Z 208.495,A -85,B 0,C 180,E1 -12773.442,E2 -12773.442} C_VEL
LIN {X 0,Y 369.316,Z 208.481,A -85,B 0,C 180,E1 -12777.819,E2 -12777.819} C_VEL
LIN {X 0,Y 369.457,Z 208.464,A -85,B 0,C 180,E1 -12780,E2 -12780} C_VEL
LIN {X 0,Y 369.317,Z 208.481,A -85,B 0,C 180,E1 -12782.181,E2 -12782.181} C_VEL
LIN {X 0,Y 369.174,Z 208.498,A -85,B 0,C 180,E1 -12786.559,E2 -12786.559} C_VEL
LIN {X 0,Y 369.063,Z 208.516,A -85,B 0,C 180,E1 -12789.868,E2 -12789.868} C_VEL
LIN {X 0,Y 369.036,Z 208.523,A -85,B 0,C 180,E1 -12793.772,E2 -12793.772} C_VEL
LIN {X 0,Y 369.026,Z 208.524,A -85,B 0,C 180,E1 -12795.322,E2 -12795.322} C_VEL
LIN {X 0,Y 370.135,Z 211.537,A -85,B 0,C 180,E1 -12795.511,E2 -12795.511} C_VEL
LIN {X 0,Y 377.036,Z 226.064,A -85,B 0,C 180,E1 -12796.413,E2 -12796.413} C_VEL
LIN {X 0,Y 379.125,Z 231.318,A -85,B 0,C 180,E1 -12796.697,E2 -12796.697} C_VEL
LIN {X 0,Y 376.969,Z 315.594,A -85,B 0,C 180,E1 -12798.566,E2 -12798.566} C_VEL
LIN {X 0,Y 376.532,Z 328.78,A -85,B 0,C 180,E1 -12799.083,E2 -12799.083} C_VEL
LIN {X 0,Y 375.855,Z 341.161,A -85,B 0,C 180,E1 -12799.78,E2 -12799.78} C_VEL
LIN {X 0,Y 374.955,Z 353.061,A -85,B 0,C 180,E1 -12800.683,E2 -12800.683} C_VEL
LIN {X 0,Y 373.98,Z 364.382,A -85,B 0,C 180,E1 -12801.787,E2 -12801.787} C_VEL
LIN {X 0,Y 373.012,Z 373.788,A -85,B 0,C 180,E1 -12802.924,E2 -12802.924} C_VEL
LIN {X 0,Y 372.034,Z 382.768,A -85,B 0,C 180,E1 -12804.26,E2 -12804.26} C_VEL
LIN {X 0,Y 371.003,Z 391.309,A -85,B 0,C 180,E1 -12805.829,E2 -12805.829} C_VEL
LIN {X 0,Y 370.129,Z 398.276,A -85,B 0,C 180,E1 -12807.417,E2 -12807.417} C_VEL
LIN {X 0,Y 369.371,Z 404.649,A -85,B 0,C 180,E1 -12809.26,E2 -12809.26} C_VEL
LIN {X 0,Y 368.769,Z 409.171,A -85,B 0,C 180,E1 -12810.968,E2 -12810.968} C_VEL
LIN {X 0,Y 368.261,Z 412.859,A -85,B 0,C 180,E1 -12812.891,E2 -12812.891} C_VEL
LIN {X 0,Y 367.885,Z 415.356,A -85,B 0,C 180,E1 -12814.968,E2 -12814.968} C_VEL
LIN {X 0,Y 367.696,Z 416.246,A -85,B 0,C 180,E1 -12816.605,E2 -12816.605} C_VEL
LIN {X 0,Y 367.625,Z 416.197,A -85,B 0,C 180,E1 -12818.39,E2 -12818.39} C_VEL
LIN {X 0,Y 367.683,Z 414.69,A -85,B 0,C 180,E1 -12820.533,E2 -12820.533} C_VEL
LIN {X 0,Y 367.863,Z 412.829,A -85,B 0,C 180,E1 -12821.965,E2 -12821.965} C_VEL
LIN {X 0,Y 368.117,Z 409.999,A -85,B 0,C 180,E1 -12823.491,E2 -12823.491} C_VEL
LIN {X 0,Y 368.448,Z 406.01,A -85,B 0,C 180,E1 -12825.109,E2 -12825.109} C_VEL
LIN {X 0,Y 368.914,Z 400.135,A -85,B 0,C 180,E1 -12826.936,E2 -12826.936} C_VEL
LIN {X 0,Y 369.581,Z 392.337,A -85,B 0,C 180,E1 -12828.812,E2 -12828.812} C_VEL
LIN {X 0,Y 370.369,Z 383.738,A -85,B 0,C 180,E1 -12830.443,E2 -12830.443} C_VEL
LIN {X 0,Y 371.238,Z 373.56,A -85,B 0,C 180,E1 -12831.985,E2 -12831.985} C_VEL
LIN {X 0,Y 372.049,Z 362.554,A -85,B 0,C 180,E1 -12833.317,E2 -12833.317} C_VEL
LIN {X 0,Y 372.902,Z 351.017,A -85,B 0,C 180,E1 -12834.416,E2 -12834.416} C_VEL
LIN {X 0,Y 373.676,Z 338.789,A -85,B 0,C 180,E1 -12835.324,E2 -12835.324} C_VEL
LIN {X 0,Y 374.16,Z 325.55,A -85,B 0,C 180,E1 -12836.047,E2 -12836.047} C_VEL
LIN {X 0,Y 374.597,Z 312.257,A -85,B 0,C 180,E1 -12836.536,E2 -12836.536} C_VEL
LIN {X 0,Y 376.142,Z 227.968,A -85,B 0,C 180,E1 -12838.333,E2 -12838.333} C_VEL
LIN {X 0,Y 368.91,Z 208.545,A -85,B 0,C 180,E1 -12839.134,E2 -12839.134} C_VEL
LIN {X 0,Y 368.976,Z 208.523,A -85,B 0,C 180,E1 -12841.564,E2 -12841.564} C_VEL
LIN {X 0,Y 368.999,Z 208.517,A -85,B 0,C 180,E1 -12844.02,E2 -12844.02} C_VEL
LIN {X 0,Y 368.922,Z 208.528,A -85,B 0,C 180,E1 -12847.605,E2 -12847.605} C_VEL
LIN {X 0,Y 368.955,Z 208.528,A -85,B 0,C 180,E1 -12851.106,E2 -12851.106} C_VEL
LIN {X 0,Y 368.997,Z 208.52,A -85,B 0,C 180,E1 -12854.535,E2 -12854.535} C_VEL
LIN {X 0,Y 369.006,Z 208.517,A -85,B 0,C 180,E1 -12857.907,E2 -12857.907} C_VEL
LIN {X 0,Y 369.092,Z 208.507,A -85,B 0,C 180,E1 -12861.238,E2 -12861.238} C_VEL
LIN {X 0,Y 369.132,Z 208.506,A -85,B 0,C 180,E1 -12864.538,E2 -12864.538} C_VEL
LIN {X 0,Y 369.315,Z 208.478,A -85,B 0,C 180,E1 -12867.819,E2 -12867.819} C_VEL
LIN {X 0,Y 369.454,Z 208.462,A -85,B 0,C 180,E1 -12870,E2 -12870} C_VEL
LIN {X 0,Y 369.308,Z 208.482,A -85,B 0,C 180,E1 -12872.182,E2 -12872.182} C_VEL
LIN {X 0,Y 369.175,Z 208.5,A -85,B 0,C 180,E1 -12876.559,E2 -12876.559} C_VEL
LIN {X 0,Y 369.06,Z 208.511,A -85,B 0,C 180,E1 -12879.683,E2 -12879.683} C_VEL
LIN {X 0,Y 368.407,Z 208.597,A -85,B 0,C 180,E1 -12880.594,E2 -12880.594} C_VEL
LIN {X 0,Y 365.545,Z 208.953,A -85,B 0,C 180,E1 -12882.073,E2 -12882.073} C_VEL
LIN {X 0,Y 363.107,Z 209.254,A -85,B 0,C 180,E1 -12883.27,E2 -12883.27} C_VEL
LIN {X 0,Y 362.054,Z 209.389,A -85,B 0,C 180,E1 -12884.196,E2 -12884.196} C_VEL
LIN {X 0,Y 361.966,Z 209.395,A -85,B 0,C 180,E1 -12884.51,E2 -12884.51} C_VEL
LIN {X 0,Y 361.959,Z 209.401,A -85,B 0,C 180,E1 -12888.1,E2 -12888.1} C_VEL
LIN {X 0,Y 361.863,Z 209.409,A -85,B 0,C 180,E1 -12891.655,E2 -12891.655} C_VEL
LIN {X 0,Y 361.895,Z 209.403,A -85,B 0,C 180,E1 -12895.293,E2 -12895.293} C_VEL
LIN {X 0,Y 361.857,Z 209.408,A -85,B 0,C 180,E1 -12899.074,E2 -12899.074} C_VEL
LIN {X 0,Y 361.85,Z 209.408,A -85,B 0,C 180,E1 -12902.945,E2 -12902.945} C_VEL
LIN {X 0,Y 361.869,Z 209.412,A -85,B 0,C 180,E1 -12905.637,E2 -12905.637} C_VEL
LIN {X 0,Y 361.83,Z 209.412,A -85,B 0,C 180,E1 -12909.019,E2 -12909.019} C_VEL
LIN {X 0,Y 361.836,Z 209.41,A -85,B 0,C 180,E1 -12912.829,E2 -12912.829} C_VEL
LIN {X 0,Y 361.819,Z 209.413,A -85,B 0,C 180,E1 -12915.947,E2 -12915.947} C_VEL
LIN {X 0,Y 361.815,Z 209.418,A -85,B 0,C 180,E1 -12919.249,E2 -12919.249} C_VEL
LIN {X 0,Y 361.866,Z 209.409,A -85,B 0,C 180,E1 -12922.982,E2 -12922.982} C_VEL
LIN {X 0,Y 361.861,Z 209.408,A -85,B 0,C 180,E1 -12926.631,E2 -12926.631} C_VEL
LIN {X 0,Y 361.867,Z 209.407,A -85,B 0,C 180,E1 -12929.671,E2 -12929.671} C_VEL
LIN {X 0,Y 361.866,Z 209.408,A -85,B 0,C 180,E1 -12933.468,E2 -12933.468} C_VEL
LIN {X 0,Y 361.881,Z 209.408,A -85,B 0,C 180,E1 -12937.144,E2 -12937.144} C_VEL
LIN {X 0,Y 361.907,Z 209.406,A -85,B 0,C 180,E1 -12940.723,E2 -12940.723} C_VEL
LIN {X 0,Y 361.946,Z 209.398,A -85,B 0,C 180,E1 -12944.226,E2 -12944.226} C_VEL
LIN {X 0,Y 362.002,Z 209.394,A -85,B 0,C 180,E1 -12946.528,E2 -12946.528} C_VEL
LIN {X 0,Y 362.003,Z 209.39,A -85,B 0,C 180,E1 -12949.937,E2 -12949.937} C_VEL
LIN {X 0,Y 362.127,Z 209.374,A -85,B 0,C 180,E1 -12953.313,E2 -12953.313} C_VEL
LIN {X 0,Y 362.275,Z 209.356,A -85,B 0,C 180,E1 -12957.776,E2 -12957.776} C_VEL
LIN {X 0,Y 362.203,Z 209.364,A -85,B 0,C 180,E1 -12961.112,E2 -12961.112} C_VEL
LIN {X 0,Y 362.268,Z 209.361,A -85,B 0,C 180,E1 -12962.224,E2 -12962.224} C_VEL
LIN {X 0,Y 362.125,Z 209.375,A -85,B 0,C 180,E1 -12966.687,E2 -12966.687} C_VEL
LIN {X 0,Y 362.031,Z 209.391,A -85,B 0,C 180,E1 -12970.062,E2 -12970.062} C_VEL
LIN {X 0,Y 361.983,Z 209.396,A -85,B 0,C 180,E1 -12973.887,E2 -12973.887} C_VEL
LIN {X 0,Y 361.914,Z 209.405,A -85,B 0,C 180,E1 -12978.102,E2 -12978.102} C_VEL
LIN {X 0,Y 361.857,Z 209.411,A -85,B 0,C 180,E1 -12981.655,E2 -12981.655} C_VEL
LIN {X 0,Y 361.864,Z 209.408,A -85,B 0,C 180,E1 -12985.295,E2 -12985.295} C_VEL
LIN {X 0,Y 361.858,Z 209.408,A -85,B 0,C 180,E1 -12989.074,E2 -12989.074} C_VEL
LIN {X 0,Y 361.85,Z 209.409,A -85,B 0,C 180,E1 -12992.945,E2 -12992.945} C_VEL
LIN {X 0,Y 361.87,Z 209.411,A -85,B 0,C 180,E1 -12995.637,E2 -12995.637} C_VEL
LIN {X 0,Y 361.828,Z 209.413,A -85,B 0,C 180,E1 -12999.018,E2 -12999.018} C_VEL
LIN {X 0,Y 361.833,Z 209.412,A -85,B 0,C 180,E1 -13002.83,E2 -13002.83} C_VEL
LIN {X 0,Y 361.815,Z 209.413,A -85,B 0,C 180,E1 -13005.947,E2 -13005.947} C_VEL
LIN {X 0,Y 361.815,Z 209.418,A -85,B 0,C 180,E1 -13009.249,E2 -13009.249} C_VEL
LIN {X 0,Y 361.865,Z 209.411,A -85,B 0,C 180,E1 -13012.981,E2 -13012.981} C_VEL
LIN {X 0,Y 361.86,Z 209.409,A -85,B 0,C 180,E1 -13016.631,E2 -13016.631} C_VEL
LIN {X 0,Y 361.921,Z 209.505,A -85,B 0,C 180,E1 -13018.484,E2 -13018.484} C_VEL
LIN {X 0,Y 364.999,Z 224.063,A -85,B 0,C 180,E1 -13021.793,E2 -13021.793} C_VEL
LIN {X 0,Y 366.08,Z 230.421,A -85,B 0,C 180,E1 -13023.182,E2 -13023.182} C_VEL
LIN {X 0,Y 364.802,Z 245.037,A -85,B 0,C 180,E1 -13026.135,E2 -13026.135} C_VEL
LIN {X 0,Y 363.85,Z 256.985,A -85,B 0,C 180,E1 -13028.519,E2 -13028.519} C_VEL
LIN {X 0,Y 368.574,Z 295.712,A -85,B 0,C 180,E1 -13029.635,E2 -13029.635} C_VEL
LIN {X 0,Y 367.24,Z 366.821,A -85,B 0,C 180,E1 -13031.195,E2 -13031.195} C_VEL
LIN {X 0,Y 366.518,Z 380.909,A -85,B 0,C 180,E1 -13031.736,E2 -13031.736} C_VEL
LIN {X 0,Y 365.639,Z 393.463,A -85,B 0,C 180,E1 -13032.45,E2 -13032.45} C_VEL
LIN {X 0,Y 364.712,Z 405.135,A -85,B 0,C 180,E1 -13033.343,E2 -13033.343} C_VEL
LIN {X 0,Y 363.649,Z 416.461,A -85,B 0,C 180,E1 -13034.445,E2 -13034.445} C_VEL
LIN {X 0,Y 362.71,Z 427.47,A -85,B 0,C 180,E1 -13035.807,E2 -13035.807} C_VEL
LIN {X 0,Y 362.011,Z 435.95,A -85,B 0,C 180,E1 -13037.099,E2 -13037.099} C_VEL
LIN {X 0,Y 361.452,Z 443.586,A -85,B 0,C 180,E1 -13038.504,E2 -13038.504} C_VEL
LIN {X 0,Y 360.91,Z 451.064,A -85,B 0,C 180,E1 -13040.189,E2 -13040.189} C_VEL
LIN {X 0,Y 360.682,Z 456.122,A -85,B 0,C 180,E1 -13041.596,E2 -13041.596} C_VEL
LIN {X 0,Y 360.569,Z 461.01,A -85,B 0,C 180,E1 -13043.284,E2 -13043.284} C_VEL
LIN {X 0,Y 360.574,Z 464.724,A -85,B 0,C 180,E1 -13044.968,E2 -13044.968} C_VEL
LIN {X 0,Y 360.551,Z 467.359,A -85,B 0,C 180,E1 -13046.647,E2 -13046.647} C_VEL
LIN {X 0,Y 360.669,Z 468.585,A -85,B 0,C 180,E1 -13047.766,E2 -13047.766} C_VEL
LIN {X 0,Y 360.656,Z 469.348,A -85,B 0,C 180,E1 -13048.883,E2 -13048.883} C_VEL
LIN {X 0,Y 360.674,Z 469.674,A -85,B 0,C 180,E1 -13050,E2 -13050} C_VEL
LIN {X 0,Y 360.633,Z 469.589,A -85,B 0,C 180,E1 -13051.116,E2 -13051.116} C_VEL
LIN {X 0,Y 360.651,Z 469.103,A -85,B 0,C 180,E1 -13052.233,E2 -13052.233} C_VEL
LIN {X 0,Y 360.507,Z 468.159,A -85,B 0,C 180,E1 -13053.353,E2 -13053.353} C_VEL
LIN {X 0,Y 360.489,Z 466.79,A -85,B 0,C 180,E1 -13054.472,E2 -13054.472} C_VEL
LIN {X 0,Y 360.419,Z 464.195,A -85,B 0,C 180,E1 -13056.024,E2 -13056.024} C_VEL
LIN {X 0,Y 360.604,Z 460.016,A -85,B 0,C 180,E1 -13057.841,E2 -13057.841} C_VEL
LIN {X 0,Y 360.868,Z 454.956,A -85,B 0,C 180,E1 -13059.528,E2 -13059.528} C_VEL
LIN {X 0,Y 361.359,Z 448.634,A -85,B 0,C 180,E1 -13061.215,E2 -13061.215} C_VEL
LIN {X 0,Y 362.262,Z 440.824,A -85,B 0,C 180,E1 -13062.891,E2 -13062.891} C_VEL
LIN {X 0,Y 363.081,Z 432.882,A -85,B 0,C 180,E1 -13064.288,E2 -13064.288} C_VEL
